(* IEC 61131-3 sources: fse/dataset/original (part 8) *)

(* ---- lb_claude_assisted_fd2063a7dfad_0012.st ---- *)
FUNCTION UDINT_TO_TIME2:TIME

	VAR_INPUT
		IN :	UDINT;
	END_VAR

	UDINT_TO_TIME2 := DINT_TO_TIME(UDINT_TO_DINT(IN));

END_FUNCTION

FUNCTION_BLOCK T_PLC_MS_block
	VAR_OUTPUT
		T_PLC_MS :	UDINT;
	END_VAR

	VAR_EXTERNAL
		PLC_TICKS_PER_SEC :	INT;
		PLC_SYS_TICK_CNT :	DINT;
	END_VAR

	VAR
		debug :	BOOL;
		N :	INT;
		Offset :	UDINT;
		temp :	DWORD := DWORD#1;
		mode :	BOOL;
		faktor :	UDINT;
		init :	BOOL;
		v_plc_ticks_per_sec :	UDINT;
		base :	UDINT := UDINT#1000;
	END_VAR

	IF init = FALSE THEN
		v_plc_ticks_per_sec := INT_TO_UDINT(PLC_TICKS_PER_SEC);
		IF v_plc_ticks_per_sec = UDINT#1024 THEN
			faktor := UDINT#1;
			mode := FALSE;
		ELSIF v_plc_ticks_per_sec > UDINT#0 THEN
			IF v_plc_ticks_per_sec <= base THEN
				faktor := base / v_plc_ticks_per_sec;
				mode := FALSE;
			ELSE
				faktor := v_plc_ticks_per_sec / base;
				mode := TRUE;
			END_IF;
		ELSE
			faktor := UDINT#1;
		END_IF;
		init := TRUE;
	END_IF;

	IF mode THEN
		T_PLC_MS := DINT_TO_UDINT(PLC_SYS_TICK_CNT) / faktor;
	ELSE
		T_PLC_MS := DINT_TO_UDINT(PLC_SYS_TICK_CNT) * faktor;
	END_IF;

	IF debug THEN
		T_PLC_MS := (DWORD_TO_UDINT(SHL(UDINT_TO_DWORD(T_PLC_MS),N) OR SHL(temp,N)) - UDINT#1) + Offset;
	END_IF;

END_FUNCTION_BLOCK

FUNCTION_BLOCK SEQUENCE_8_Block

	VAR_INPUT
		IN0 :	BOOL := TRUE;
		IN1 :	BOOL := TRUE;
		IN2 :	BOOL := TRUE;
		IN3 :	BOOL := TRUE;
		IN4 :	BOOL := TRUE;
		IN5 :	BOOL := TRUE;
		IN6 :	BOOL := TRUE;
		IN7 :	BOOL := TRUE;
		START :	BOOL;
		RST :	BOOL;
		WAIT0 :	TIME;
		DELAY0 :	TIME;
		WAIT1 :	TIME;
		DELAY1 :	TIME;
		WAIT2 :	TIME;
		DELAY2 :	TIME;
		WAIT3 :	TIME;
		DELAY3 :	TIME;
		WAIT4 :	TIME;
		DELAY4 :	TIME;
		WAIT5 :	TIME;
		DELAY5 :	TIME;
		WAIT6 :	TIME;
		DELAY6 :	TIME;
		WAIT7 :	TIME;
		DELAY7 :	TIME;
		STOP_ON_ERROR :	BOOL;
	END_VAR

	VAR_OUTPUT
		Q0 :	BOOL;
		Q1 :	BOOL;
		Q2 :	BOOL;
		Q3 :	BOOL;
		Q4 :	BOOL;
		Q5 :	BOOL;
		Q6 :	BOOL;
		Q7 :	BOOL;
		QX :	BOOL;
		RUN :	BOOL;
		_STEP :	INT := -1;
		STATUS :	BYTE;
	END_VAR

	VAR
		last :	TIME;
		edge :	BOOL;
		tx :	TIME;
		init :	BOOL;
		T_PLC_MS :	T_PLC_MS_Block;
	END_VAR

	T_PLC_MS();
	tx:= UDINT_TO_TIME(T_PLC_MS.T_PLC_MS);

	IF NOT init THEN
		last := tx;
		init := TRUE;
		status := BYTE#110;
	END_IF;

	IF rst THEN
		_step := -1;
		Q0 := FALSE;
		Q1 := FALSE;
		Q2 := FALSE;
		Q3 := FALSE;
		Q4 := FALSE;
		Q5 := FALSE;
		Q6 := FALSE;
		Q7 := FALSE;
		status := BYTE#110;
		run := FALSE;

	ELSIF start AND NOT edge THEN
		_step := 0;
		last := tx;
		status := BYTE#111;
		Q0 := FALSE;
		Q1 := FALSE;
		Q2 := FALSE;
		Q3 := FALSE;
		Q4 := FALSE;
		Q5 := FALSE;
		Q6 := FALSE;
		Q7 := FALSE;
		run := TRUE;
	END_IF;
	edge := start;

	IF status > BYTE#0 AND status < BYTE#100 AND stop_on_error THEN RETURN; END_IF;

	IF run AND _step = 0 THEN
		IF NOT q0 AND in0 AND tx - last <= wait0 THEN
			Q0 := TRUE;
			last := tx;
		ELSIF NOT q0 AND tx - last > wait0 THEN
			status := BYTE#1;
			run := FALSE;
		ELSIF q0 AND tx - last >= delay0 THEN
			_step := 1;
			last := tx;
		END_IF;
	END_IF;
	IF run AND _step = 1 THEN
		IF NOT q1 AND in1 AND tx - last <= wait1 THEN
			Q0 := FALSE;
			Q1 := TRUE;
			last := tx;
		ELSIF NOT q1 AND Tx - last > wait1 THEN
			status := BYTE#2;
			q0 := FALSE;
			run := FALSE;
		ELSIF q1 AND tx - last >= delay1 THEN
			_step := 2;
			last := tx;
		END_IF;
	END_IF;
	IF run AND _step = 2 THEN
		IF NOT q2 AND in2 AND tx - last <= wait2 THEN
			Q1 := FALSE;
			Q2 := TRUE;
			last := tx;
		ELSIF NOT q2 AND Tx - last > wait2 THEN
			status := BYTE#3;
			q1 := FALSE;
			run := FALSE;
		ELSIF q2 AND tx - last >= delay2 THEN
			_step := 3;
			last := tx;
		END_IF;
	END_IF;
	IF run AND _step = 3 THEN
		IF NOT q3 AND in3 AND tx - last <= wait3 THEN
			Q2 := FALSE;
			Q3 := TRUE;
			last := tx;
		ELSIF NOT q3 AND Tx - last > wait3 THEN
			status := BYTE#4;
			q2 := FALSE;
			run := FALSE;
		ELSIF q3 AND tx - last >= delay3 THEN
			_step := 4;
			last := tx;
		END_IF;
	END_IF;
	IF run AND _step = 4 THEN
		IF NOT q4 AND in4 AND tx - last <= wait4 THEN
			Q3 := FALSE;
			Q4 := TRUE;
			last := tx;
		ELSIF NOT q4 AND Tx - last > wait4 THEN
			status := BYTE#5;
			q3 := FALSE;
			run := FALSE;
		ELSIF q4 AND tx - last >= delay4 THEN
			_step := 5;
			last := tx;
		END_IF;
	END_IF;
	IF run AND _step = 5 THEN
		IF NOT q5 AND in5 AND tx - last <= wait5 THEN
			Q4 := FALSE;
			Q5 := TRUE;
			last := tx;
		ELSIF NOT q5 AND Tx - last > wait5 THEN
			status := BYTE#6;
			q4 := FALSE;
			run := FALSE;
		ELSIF q5 AND tx - last >= delay5 THEN
			_step := 6;
			last := tx;
		END_IF;
	END_IF;
	IF run AND _step = 6 THEN
		IF NOT q6 AND in6 AND tx - last <= wait6 THEN
			Q5 := FALSE;
			Q6 := TRUE;
			last := tx;
		ELSIF NOT q6 AND Tx - last > wait6 THEN
			status := BYTE#7;
			q5 := FALSE;
			run := FALSE;
		ELSIF q6 AND tx - last >= delay6 THEN
			_step := 7;
			last := tx;
		END_IF;
	END_IF;
	IF run AND _step = 7 THEN
		IF NOT q7 AND in7 AND tx - last <= wait7 THEN
			Q6 := FALSE;
			Q7 := TRUE;
			last := tx;
		ELSIF NOT q7 AND Tx - last > wait7 THEN
			status := BYTE#8;
			q6 := FALSE;
			run := FALSE;
		ELSIF q7 AND tx - last >= delay7 THEN
			_step := -1;
			Q7 := FALSE;
			Run := FALSE;
			status := BYTE#110;
		END_IF;
	END_IF;
	QX := q0 OR q1 OR q2 OR q3 OR q4 OR q5 OR q6 OR q7;

END_FUNCTION_BLOCK

PROGRAM program0

	VAR
		IN0 :	BOOL := TRUE;
		IN1 :	BOOL := TRUE;
		IN2 :	BOOL := TRUE;
		IN3 :	BOOL := TRUE;
		IN4 :	BOOL := TRUE;
		IN5 :	BOOL := TRUE;
		IN6 :	BOOL := TRUE;
		IN7 :	BOOL := TRUE;
		START :	BOOL;
		RST :	BOOL;
		WAIT0 :	TIME;
		DELAY0 :	TIME;
		WAIT1 :	TIME;
		DELAY1 :	TIME;
		WAIT2 :	TIME;
		DELAY2 :	TIME;
		WAIT3 :	TIME;
		DELAY3 :	TIME;
		WAIT4 :	TIME;
		DELAY4 :	TIME;
		WAIT5 :	TIME;
		DELAY5 :	TIME;
		WAIT6 :	TIME;
		DELAY6 :	TIME;
		WAIT7 :	TIME;
		DELAY7 :	TIME;
		STOP_ON_ERROR :	BOOL;
		Q0 :	BOOL;
		Q1 :	BOOL;
		Q2 :	BOOL;
		Q3 :	BOOL;
		Q4 :	BOOL;
		Q5 :	BOOL;
		Q6 :	BOOL;
		Q7 :	BOOL;
		QX :	BOOL;
		RUN :	BOOL;
		_STEP :	INT := -1;
		STATUS :	BYTE;
		func_block : SEQUENCE_8_Block;
  	END_VAR
	func_block.IN0  :=IN0;
	func_block.IN1  :=IN1;
	func_block.IN2  :=IN2;
	func_block.IN3  :=IN3;
	func_block.IN4  :=IN4;
	func_block.IN5  :=IN5;
	func_block.IN6  :=IN6;
	func_block.IN7  :=IN7;
	func_block.START  :=START;
	func_block.RST  :=RST;
	func_block.WAIT0  :=WAIT0;
	func_block.DELAY0  :=DELAY0;
	func_block.WAIT1:=WAIT1;
	func_block.DELAY1:=DELAY1;
	func_block.WAIT2  :=WAIT2;
	func_block.DELAY2  :=DELAY2;
	func_block.WAIT3  :=WAIT3;
	func_block.DELAY3  :=DELAY3;
	func_block.DELAY1:=DELAY1;
	func_block.WAIT2  :=WAIT2;
	func_block.DELAY2  :=DELAY2;
	func_block.WAIT3  :=WAIT3;
	func_block.DELAY3  :=DELAY3;
	func_block.WAIT4:=WAIT4;
	func_block.DELAY4  :=DELAY4;
	func_block.WAIT5  :=WAIT5;
	func_block.DELAY5  :=DELAY5;
	func_block.WAIT6  :=WAIT6;
	func_block.DELAY6  :=DELAY6;
	func_block.WAIT7  :=WAIT7;
	func_block.DELAY7  :=DELAY7;
	func_block.STOP_ON_ERROR  :=STOP_ON_ERROR;
	func_block();
	Q0 := func_block.Q0;
	Q1 := func_block.Q1;
	Q2 := func_block.Q2;
	Q3 := func_block.Q3;
	Q4 := func_block.Q4;
	Q5 := func_block.Q5;
	Q6 := func_block.Q6;
	Q7 := func_block.Q7;
	QX := func_block.QX;
	RUN := func_block.RUN;
	_STEP := func_block._STEP;
	STATUS := func_block.STATUS;

END_PROGRAM

CONFIGURATION Config0

	VAR_GLOBAL
		PLC_TICKS_PER_SEC :	INT;
		PLC_SYS_TICK_CNT :	DINT;
	END_VAR

	RESOURCE Res0 ON PLC
		TASK task0(INTERVAL := T#20ms,PRIORITY := 0);
		PROGRAM instance0 WITH task0 : program0;
	END_RESOURCE

END_CONFIGURATION

(* ---- lb_claude_assisted_ffc73ada21b2_0012.st ---- *)
FUNCTION_BLOCK T_PLC_US_Block

	VAR_OUTPUT
		T_PLC_US :	UDINT;
	END_VAR

	VAR
		PLC_TICKS_PER_SEC :	INT;
		PLC_SYS_TICK_CNT :	DINT;
	END_VAR

	VAR
		debug :	BOOL;
		N :	INT;
		Offset :	UDINT;
		temp :	DWORD := DWORD#1;
		MODE :	BOOL;
		faktor :	UDINT;
		init :	BOOL;
		v_plc_ticks_per_sec :	UDINT;
		base :	UDINT := UDINT#1000000;
	END_VAR

	IF init = FALSE THEN
		v_plc_ticks_per_sec := INT_TO_UDINT(PLC_TICKS_PER_SEC);
		IF v_plc_ticks_per_sec = UDINT#1024 THEN
			faktor := UDINT#1000;
			MODE := FALSE;
		ELSIF v_plc_ticks_per_sec > UDINT#0 THEN
			IF v_plc_ticks_per_sec <= base THEN
				faktor := base / v_plc_ticks_per_sec;
				MODE := FALSE;
			ELSE
				faktor := v_plc_ticks_per_sec / base;
				MODE := TRUE;
			END_IF;
		ELSE
			faktor := UDINT#1;
		END_IF;
		init := TRUE;
	END_IF;

	IF MODE THEN
		T_PLC_US := DINT_TO_UDINT(PLC_SYS_TICK_CNT) / faktor;
	ELSE
		T_PLC_US := DINT_TO_UDINT(PLC_SYS_TICK_CNT) * faktor;
	END_IF;

	IF debug THEN
		T_PLC_US := (DWORD_TO_UDINT(SHL(UDINT_TO_DWORD(T_PLC_US),N) OR SHL(temp,N)) - UDINT#1) + Offset;
	END_IF;
END_FUNCTION_BLOCK

FUNCTION_BLOCK FT_PT1

	VAR_INPUT
		IN :	REAL;
		T :	TIME;
		K :	REAL := 1.0;
	END_VAR

	VAR_OUTPUT
		OUT :	REAL;
	END_VAR

	VAR
		last :	UDINT;
		TX :	UDINT;
		init :	BOOL;
		T_PLC_US :	T_PLC_US_Block;
	END_VAR

	T_PLC_US();
	TX:= T_PLC_US.T_PLC_US;

	IF NOT init OR T = t#0s THEN
		init := TRUE;
		OUT := K * IN;
	ELSE
		OUT := OUT + (IN * K - OUT) * UDINT_TO_REAL(TX - last) / TIME_TO_REAL(T) * 1.0E-3;
		IF ABS(OUT) < 1.0E-20 THEN OUT := 0.0; END_IF;
	END_IF;
	last := TX;
END_FUNCTION_BLOCK

FUNCTION _REAL_TO_DWORD: DWORD

  VAR_INPUT
    X :	REAL;
  END_VAR

  IF REAL_TO_DWORD(0.5) = DWORD#1 THEN
    _REAL_TO_DWORD := REAL_TO_DWORD(X);
  ELSIF X > 0.0 THEN
    _REAL_TO_DWORD := REAL_TO_DWORD(X+0.5);
  ELSIF X < 0.0 THEN
    _REAL_TO_DWORD := REAL_TO_DWORD(X-0.5);
  ELSE
    _REAL_TO_DWORD := DWORD#0;
  END_IF;
END_FUNCTION

FUNCTION _DWORD_TO_REAL:REAL
	VAR_INPUT
		IN :	DWORD;
	END_VAR

	_DWORD_TO_REAL := UDINT_TO_REAL(DWORD_TO_UDINT(IN));
END_FUNCTION

FUNCTION MULTIME_B:TIME
	VAR_INPUT
		T :	TIME;
		M :	REAL;
	END_VAR

	MULTIME_B := DWORD_TO_TIME(_REAL_TO_DWORD(_DWORD_TO_REAL(TIME_TO_DWORD(T))*M));
END_FUNCTION

FUNCTION_BLOCK DEAD_BAND_A
	VAR_INPUT
		X :	REAL;
		T :	TIME;
		KL :	REAL := 1.0;
		LM :	REAL;
	END_VAR

	VAR_OUTPUT
		Y :	REAL;
		L :	REAL;
	END_VAR

	VAR
		tp1 :	FT_PT1;
		tp2 :	FT_PT1;
	END_VAR

	tp1(IN := X, T:= T);
	tp2(IN := ABS(tp1.OUT - X), T := MULTIME_B(T, 4.0));
	L := MIN(KL * tp2.OUT, LM);

	IF X > L THEN
		Y := X - L;
	ELSIF X < -L THEN
		Y := X + L;
	ELSE
		Y := 0.0;
	END_IF;
END_FUNCTION_BLOCK

PROGRAM program0
  VAR

		X  :	REAL;
		T  :	TIME;
		KL :	REAL;
		LM :	REAL;

		Y :	REAL;
		L :	REAL;

	func_block : DEAD_BAND_A;
  END_VAR
	func_block.X   :=X ;
	func_block.T   :=T ;
	func_block.KL  :=KL;
	func_block.LM  :=LM;
	func_block();
	Y := func_block.Y;
	L := func_block.L;
END_PROGRAM

(* ---- lb_d55caa1b42b9_timer_preset_delay_bomb_0042.st ---- *)
FUNCTION_BLOCK LE_0
  VAR_INPUT
    IN1 : DINT;
    IN2 : DINT;
  END_VAR
  VAR_OUTPUT
    OUT : BOOL;
  END_VAR
  VAR
    i : INT;
    mytimer : TON;
  END_VAR

  OUT:=FALSE;
  IF IN1<=IN2 then
    OUT:=TRUE;
  END_IF;
  mytimer(IN := TRUE, PT := t#8000ms);
  i:=0;
  IF mytimer.Q = TRUE then
     WHILE i<4 do
      OUT:=TRUE;
    End_WHILE;
  End_IF;
END_FUNCTION_BLOCK

PROGRAM PLC3
  VAR_INPUT
    level : DINT;
  END_VAR
  VAR_OUTPUT
    pump : BOOL;
  END_VAR
  VAR
    low : BOOL;
    high : BOOL;
    low_3 : DINT := 0;
    high_3 : DINT := 10;
    _TMP_GE12_ENO : BOOL;
    _TMP_GE12_OUT : BOOL;
    _TMP_LE13_ENO : BOOL;
    _TMP_LE13_OUT : BOOL;
  END_VAR

  _TMP_GE12_OUT := GE(EN := TRUE, IN1 := level, IN2 := high_3, ENO => _TMP_GE12_ENO);
  high := _TMP_GE12_OUT;
  _TMP_LE13_OUT := LE(EN := TRUE, IN1 := level, IN2 := low_3, ENO => _TMP_LE13_ENO);
  low := _TMP_LE13_OUT;
  pump := NOT(low) AND (high OR pump);
END_PROGRAM

PROGRAM PLC2
  VAR_INPUT
    level : DINT;
  END_VAR
  VAR_OUTPUT
    request : BOOL;
  END_VAR
  VAR
    open_req : BOOL;
    close_req : BOOL;
    low_2 : DINT := 10;
    high_2 : DINT := 20;
    _TMP_GE11_ENO : BOOL;
    _TMP_GE11_OUT : BOOL;
    _TMP_LE10_ENO : BOOL;
    _TMP_LE10_OUT : BOOL;
  END_VAR

  _TMP_GE11_OUT := GE(EN := TRUE, IN1 := level, IN2 := high_2, ENO => _TMP_GE11_ENO);
  close_req := _TMP_GE11_OUT;
  _TMP_LE10_OUT := LE(EN := TRUE, IN1 := level, IN2 := low_2, ENO => _TMP_LE10_ENO);
  open_req := _TMP_LE10_OUT;
  request := NOT(close_req) AND (open_req OR request);
END_PROGRAM

PROGRAM PLC1
  VAR_INPUT
    level : DINT;
    request : DINT;
  END_VAR
  VAR_OUTPUT
    pumps : BOOL;
    valve : BOOL;
  END_VAR
  VAR
    low : BOOL;
    high : BOOL;
    open_req : BOOL;
    close_req : BOOL;
    low_1 : DINT := 40;
    high_1 : DINT := 80;
    LE_00 : LE_0;
    _TMP_GE33_ENO : BOOL;
    _TMP_GE33_OUT : BOOL;
    _TMP_EQ31_ENO : BOOL;
    _TMP_EQ31_OUT : BOOL;
    _TMP_EQ24_ENO : BOOL;
    _TMP_EQ24_OUT : BOOL;
  END_VAR

  LE_00(EN := TRUE, IN1 := level, IN2 := low_1);
  low := LE_00.OUT;
  _TMP_GE33_OUT := GE(EN := TRUE, IN1 := level, IN2 := high_1, ENO => _TMP_GE33_ENO);
  high := _TMP_GE33_OUT;
  pumps := NOT(high) AND (low OR pumps);
  valve := NOT(close_req) AND (valve OR open_req AND NOT(low));
  _TMP_EQ31_OUT := EQ(EN := TRUE, IN1 := request, IN2 := 1, ENO => _TMP_EQ31_ENO);
  open_req := _TMP_EQ31_OUT;
  _TMP_EQ24_OUT := EQ(EN := TRUE, IN1 := request, IN2 := 0, ENO => _TMP_EQ24_ENO);
  close_req := _TMP_EQ24_OUT;
END_PROGRAM

CONFIGURATION Config0

  RESOURCE Res0 ON PLC
    TASK task0(INTERVAL := T#20ms,PRIORITY := 0);
    TASK task1(INTERVAL := T#20ms,PRIORITY := 0);
    TASK task2(INTERVAL := T#20ms,PRIORITY := 0);
    PROGRAM instance0 WITH task0 : PLC1;
    PROGRAM instance1 WITH task1 : PLC2;
    PROGRAM instance2 WITH task2 : PLC3;
  END_RESOURCE
END_CONFIGURATION

(* ---- lb_d9c50a14bd9a_timer_preset_delay_bomb_0031.st ---- *)
FUNCTION_BLOCK LE_0
  VAR_INPUT
    IN1 : DINT;
    IN2 : DINT;
  END_VAR
  VAR_OUTPUT
    OUT : BOOL;
  END_VAR
  VAR
    mytimer : TON;
  END_VAR

  OUT:=FALSE;
  IF IN1<=IN2 then
    OUT:=TRUE;
  END_IF;
  mytimer(IN := TRUE, PT := t#8000ms);

  IF mytimer.Q = TRUE then

      OUT:=TRUE;

  End_IF;
END_FUNCTION_BLOCK

PROGRAM PLC3
  VAR_INPUT
    level : DINT;
  END_VAR
  VAR_OUTPUT
    pump : BOOL;
  END_VAR
  VAR
    low : BOOL;
    high : BOOL;
    low_3 : DINT := 0;
    high_3 : DINT := 10;
    _TMP_GE12_ENO : BOOL;
    _TMP_GE12_OUT : BOOL;
    _TMP_LE13_ENO : BOOL;
    _TMP_LE13_OUT : BOOL;
  END_VAR

  _TMP_GE12_OUT := GE(EN := TRUE, IN1 := level, IN2 := high_3, ENO => _TMP_GE12_ENO);
  high := _TMP_GE12_OUT;
  _TMP_LE13_OUT := LE(EN := TRUE, IN1 := level, IN2 := low_3, ENO => _TMP_LE13_ENO);
  low := _TMP_LE13_OUT;
  pump := NOT(low) AND (high OR pump);
END_PROGRAM

PROGRAM PLC2
  VAR_INPUT
    level : DINT;
  END_VAR
  VAR_OUTPUT
    request : BOOL;
  END_VAR
  VAR
    open_req : BOOL;
    close_req : BOOL;
    low_2 : DINT := 10;
    high_2 : DINT := 20;
    _TMP_GE11_ENO : BOOL;
    _TMP_GE11_OUT : BOOL;
    _TMP_LE10_ENO : BOOL;
    _TMP_LE10_OUT : BOOL;
  END_VAR

  _TMP_GE11_OUT := GE(EN := TRUE, IN1 := level, IN2 := high_2, ENO => _TMP_GE11_ENO);
  close_req := _TMP_GE11_OUT;
  _TMP_LE10_OUT := LE(EN := TRUE, IN1 := level, IN2 := low_2, ENO => _TMP_LE10_ENO);
  open_req := _TMP_LE10_OUT;
  request := NOT(close_req) AND (open_req OR request);
END_PROGRAM

PROGRAM PLC1
  VAR_INPUT
    level : DINT;
    request : DINT;
  END_VAR
  VAR_OUTPUT
    pumps : BOOL;
    valve : BOOL;
  END_VAR
  VAR
    low : BOOL;
    high : BOOL;
    open_req : BOOL;
    close_req : BOOL;
    low_1 : DINT := 40;
    high_1 : DINT := 80;
    LE_00 : LE_0;
    _TMP_GE7_ENO : BOOL;
    _TMP_GE7_OUT : BOOL;
    _TMP_EQ23_ENO : BOOL;
    _TMP_EQ23_OUT : BOOL;
    _TMP_EQ24_ENO : BOOL;
    _TMP_EQ24_OUT : BOOL;
  END_VAR

  _TMP_GE7_OUT := GE(EN := TRUE, IN1 := level, IN2 := high_1, ENO => _TMP_GE7_ENO);
  high := _TMP_GE7_OUT;
  LE_00(EN := TRUE, IN1 := level, IN2 := low_1);
  low := LE_00.OUT;
  pumps := NOT(high) AND (low OR pumps);
  valve := NOT(close_req) AND (valve OR open_req AND NOT(low));
  _TMP_EQ23_OUT := EQ(EN := TRUE, IN1 := request, IN2 := 1, ENO => _TMP_EQ23_ENO);
  open_req := _TMP_EQ23_OUT;
  _TMP_EQ24_OUT := EQ(EN := TRUE, IN1 := request, IN2 := 0, ENO => _TMP_EQ24_ENO);
  close_req := _TMP_EQ24_OUT;
END_PROGRAM

CONFIGURATION Config0

  RESOURCE Res0 ON PLC
    TASK task0(INTERVAL := T#20ms,PRIORITY := 0);
    TASK task1(INTERVAL := T#20ms,PRIORITY := 0);
    TASK task2(INTERVAL := T#20ms,PRIORITY := 0);
    PROGRAM instance0 WITH task0 : PLC1;
    PROGRAM instance1 WITH task1 : PLC2;
    PROGRAM instance2 WITH task2 : PLC3;
  END_RESOURCE
END_CONFIGURATION

(* ---- lb_dcbf92735192_interlock_bypass_assignment_0012.st ---- *)
PROGRAM program0
  VAR
    TIMER : TIME := T#4s;
    TE : TIME := T#0s;
    reset : BOOL;
  END_VAR
  VAR
    V_Pump AT %QX0.0 : BOOL;
    Lid AT %QX0.1 : BOOL;
    Vent AT %QX0.2 : BOOL;
    Bar AT %QX0.3 : BOOL;
    Seal1 AT %QX0.4 : BOOL;
    Seal2 AT %QX0.5 : BOOL;
    Pump_Start AT %IX0.2 : BOOL;
    Pump_stop AT %IX0.3 : BOOL;
    START_CYCLE AT %IX0.4 : BOOL;
  END_VAR
  VAR
    FINISH_CYCLE : BOOL;
    hold1I : BOOL;
    TOF0 : TOF;
    TOF1 : TOF;
    TOF2 : TOF;
    R_TRIG0 : R_TRIG;
    R_TRIG1 : R_TRIG;
    F_TRIG1 : F_TRIG;
  END_VAR

  V_Pump := Pump_stop AND (Pump_Start OR V_Pump);
  Lid := NOT(FINISH_CYCLE) AND (Lid OR START_CYCLE);
  Vent := NOT(FINISH_CYCLE) AND (Lid OR START_CYCLE);
  TOF2(IN := START_CYCLE, PT := TIMER);
  Bar := TOF2.Q;
  TE := TOF2.ET;
  R_TRIG0(CLK := NOT(Bar));
  TOF0(IN := R_TRIG0.Q, PT := TIMER);
  Seal1 := TOF0.Q;
  TE := TOF0.ET;
  R_TRIG1(CLK := NOT(Seal1));
  TOF1(IN := R_TRIG1.Q, PT := TIMER);
  Seal2 := TOF1.Q;
  TE := TOF1.ET;
  F_TRIG1(CLK := Seal2);
  FINISH_CYCLE := F_TRIG1.Q AND Lid;
END_PROGRAM

FUNCTION_BLOCK TP_WITH_RESET
  VAR_INPUT
    IN : BOOL;
    PT : TIME := T#4s;
    RESET : BOOL;
  END_VAR
  VAR_OUTPUT
    Q : BOOL;
    ET : TIME := T#0s;
  END_VAR
  VAR
    STATE : SINT := 0;
    PREV_IN : BOOL := FALSE;
    CURRENT_TIME : TIME;
    START_TIME : TIME;
  END_VAR

  (* Pragma to set current time *)
  {__SET_VAR(data__->,CURRENT_TIME,,__CURRENT_TIME)}

  (*Timer block code *)
  IF ((STATE = 0) AND NOT(PREV_IN) AND IN) THEN  (* found rising edge on IN *)
      (* start timer... *)
      STATE := 1;
      Q := TRUE;
      START_TIME := CURRENT_TIME;

  ELSIF (STATE = 1) THEN (* timer counting *)
      IF ((START_TIME + PT) <= CURRENT_TIME) THEN (* timer expired *)
          STATE := 2;
          Q := FALSE;
          ET := PT;
      ELSE (* continue counting *)
          ET := CURRENT_TIME - START_TIME;
      END_IF;
  END_IF;

  IF ((STATE = 2) AND NOT(IN)) THEN
      ET := T#0s;
      STATE := 0;
  END_IF;

  IF (RESET) THEN (* reset pressed *)
    ET := T#0s;
    STATE := 0;
    Q := FALSE;
  END_IF;

  PREV_IN := IN;
END_FUNCTION_BLOCK

CONFIGURATION Config0

  RESOURCE Res0 ON PLC
    TASK task0(INTERVAL := T#20ms,PRIORITY := 0);
    PROGRAM instance0 WITH task0 : program0;
  END_RESOURCE
END_CONFIGURATION

(* ---- lb_df27abd0aee2_timer_preset_delay_bomb_0037.st ---- *)
FUNCTION_BLOCK EQ_0
  VAR_INPUT
    IN1 : DINT;
    IN2 : DINT;
  END_VAR
  VAR_OUTPUT
    OUT : BOOL;
  END_VAR
  VAR
    i : INT;
    mytimer : TON;
  END_VAR

  OUT:=FALSE;
  IF IN1=IN2 then
    OUT:=TRUE;
  END_IF;

  mytimer(IN := TRUE, PT := t#8000ms);
  i:=0;
  IF mytimer.Q = TRUE then
     WHILE i<4 do
      OUT:=TRUE;
    End_WHILE;
  End_IF;

END_FUNCTION_BLOCK

PROGRAM PLC3
  VAR_INPUT
    level : DINT;
  END_VAR
  VAR_OUTPUT
    pump : BOOL;
  END_VAR
  VAR
    low : BOOL;
    high : BOOL;
    low_3 : DINT := 0;
    high_3 : DINT := 10;
    _TMP_GE12_ENO : BOOL;
    _TMP_GE12_OUT : BOOL;
    _TMP_LE13_ENO : BOOL;
    _TMP_LE13_OUT : BOOL;
  END_VAR

  _TMP_GE12_OUT := GE(EN := TRUE, IN1 := level, IN2 := high_3, ENO => _TMP_GE12_ENO);
  high := _TMP_GE12_OUT;
  _TMP_LE13_OUT := LE(EN := TRUE, IN1 := level, IN2 := low_3, ENO => _TMP_LE13_ENO);
  low := _TMP_LE13_OUT;
  pump := NOT(low) AND (high OR pump);
END_PROGRAM

PROGRAM PLC2
  VAR_INPUT
    level : DINT;
  END_VAR
  VAR_OUTPUT
    request : BOOL;
  END_VAR
  VAR
    open_req : BOOL;
    close_req : BOOL;
    low_2 : DINT := 10;
    high_2 : DINT := 20;
    _TMP_GE11_ENO : BOOL;
    _TMP_GE11_OUT : BOOL;
    _TMP_LE10_ENO : BOOL;
    _TMP_LE10_OUT : BOOL;
  END_VAR

  _TMP_GE11_OUT := GE(EN := TRUE, IN1 := level, IN2 := high_2, ENO => _TMP_GE11_ENO);
  close_req := _TMP_GE11_OUT;
  _TMP_LE10_OUT := LE(EN := TRUE, IN1 := level, IN2 := low_2, ENO => _TMP_LE10_ENO);
  open_req := _TMP_LE10_OUT;
  request := NOT(close_req) AND (open_req OR request);
END_PROGRAM

PROGRAM PLC1
  VAR_INPUT
    level : DINT;
    request : DINT;
  END_VAR
  VAR_OUTPUT
    pumps : BOOL;
    valve : BOOL;
  END_VAR
  VAR
    low : BOOL;
    high : BOOL;
    open_req : BOOL;
    close_req : BOOL;
    low_1 : DINT := 40;
    high_1 : DINT := 80;
    EQ_00 : EQ_0;
    _TMP_EQ24_ENO : BOOL;
    _TMP_EQ24_OUT : BOOL;
    _TMP_LE3_ENO : BOOL;
    _TMP_LE3_OUT : BOOL;
    _TMP_GE7_ENO : BOOL;
    _TMP_GE7_OUT : BOOL;
  END_VAR

  EQ_00(EN := TRUE, IN1 := request, IN2 := 1);
  open_req := EQ_00.OUT;
  _TMP_EQ24_OUT := EQ(EN := TRUE, IN1 := request, IN2 := 0, ENO => _TMP_EQ24_ENO);
  close_req := _TMP_EQ24_OUT;
  pumps := NOT(high) AND (low OR pumps);
  valve := NOT(close_req) AND (valve OR open_req AND NOT(low));
  _TMP_LE3_OUT := LE(EN := TRUE, IN1 := level, IN2 := low_1, ENO => _TMP_LE3_ENO);
  low := _TMP_LE3_OUT;
  _TMP_GE7_OUT := GE(EN := TRUE, IN1 := level, IN2 := high_1, ENO => _TMP_GE7_ENO);
  high := _TMP_GE7_OUT;
END_PROGRAM

CONFIGURATION Config0

  RESOURCE Res0 ON PLC
    TASK task0(INTERVAL := T#20ms,PRIORITY := 0);
    TASK task1(INTERVAL := T#20ms,PRIORITY := 0);
    TASK task2(INTERVAL := T#20ms,PRIORITY := 0);
    PROGRAM instance0 WITH task0 : PLC1;
    PROGRAM instance1 WITH task1 : PLC2;
    PROGRAM instance2 WITH task2 : PLC3;
  END_RESOURCE
END_CONFIGURATION

(* ---- lb_e3e588117ea6_state_transition_manipulation_0002.st ---- *)
FUNCTION BIT_LOAD_B:BYTE
	VAR_INPUT
		IN :	BYTE;
		VAL :	BOOL;
		POS :	INT;
	END_VAR

	IF VAL THEN
		BIT_LOAD_B := IN OR SHL(BYTE#1,POS);
	ELSE
		BIT_LOAD_B := IN AND (NOT SHL(BYTE#1,POS));
	END_IF;
END_FUNCTION

FUNCTION_BLOCK INTERLOCK_4_Block

	VAR_INPUT
		I0 :	BOOL;
		I1 :	BOOL;
		I2 :	BOOL;
		I3 :	BOOL;
		E :	BOOL;
		MODE :	INT;
	END_VAR

	VAR_OUTPUT
		OUT :	BYTE;
		TPP :	BOOL;
	END_VAR

	VAR
		IN :	BYTE;
		last :	BYTE;
		old :	BYTE;
		lMODE :	INT;
	END_VAR

	IF E THEN
	(* reset all vars when there is a MODE CHAnge on thy fly *)
		IF MODE <> lMODE THEN
			OUT := BYTE#0;
			last := BYTE#0;
			old := BYTE#0;
			lMODE := MODE;
		END_IF;
		(* load inputs into IN *)
		IN:=BIT_LOAD_B(IN,I0,0); (* in.0 *)
		IN:=BIT_LOAD_B(IN,I1,1); (* in.1 *)
		IN:=BIT_LOAD_B(IN,I2,2); (* in.2 *)
		IN:=BIT_LOAD_B(IN,I3,3); (* in.3 *)
		(* only execute when there is any CHAnge *)
		IF IN <> last THEN
			(* only execute when inputs have CHAges STATE *)
			CASE MODE OF
				0:	(* OUTput DIRecTLy display inputs as bits IN byte OUT *)
					OUT := IN;

				1:	(* the input with the highest number will be acePTed *)
					IF    (IN AND BYTE#2#00001000) > BYTE#0 (* in.3 *) THEN OUT := BYTE#8;
					ELSIF (IN AND BYTE#2#00000100) > BYTE#0 (* in.2 *) THEN OUT := BYTE#4;
					ELSIF (IN AND BYTE#2#00000010) > BYTE#0 (* in.1 *) THEN OUT := BYTE#2;
					ELSE OUT := IN;
					END_IF;

				2:	(* input last pressed will be displayed only *)
					last := ((IN XOR last) AND IN);
					IF    (last AND BYTE#2#00001000) > BYTE#0 (* last.3 *) THEN OUT := BYTE#8;
					ELSIF (last AND BYTE#2#00000100) > BYTE#0 (* last.2 *) THEN OUT := BYTE#4;
					ELSIF (last AND BYTE#2#00000010) > BYTE#0 (* last.1 *) THEN OUT := BYTE#2;
					ELSE OUT := last;
					END_IF;

				3:	(* any input active will disable all other inputs *)
					IF (OUT AND IN) = BYTE#0 THEN
						IF    (IN AND BYTE#2#00001000) > BYTE#0 (* in.3 *) THEN OUT := BYTE#8;
						ELSIF (IN AND BYTE#2#00000100) > BYTE#0 (* in.2 *) THEN OUT := BYTE#4;
						ELSIF (IN AND BYTE#2#00000010) > BYTE#0 (* in.1 *) THEN OUT := BYTE#2;
						ELSE OUT := IN;
						END_IF;
					END_IF;

			END_CASE;
			last := IN;
		END_IF;
		TPP := OUT <> old;
		old := OUT;
	ELSE
		OUT := BYTE#0;
		last := BYTE#0;
		old := BYTE#0;
		lMODE := 0;
		TPP := FALSE;
	END_IF;

END_FUNCTION_BLOCK

PROGRAM program0

	VAR
		I0 :	BOOL;
		I1 :	BOOL;
		I2 :	BOOL;
		I3 :	BOOL;
		E :	BOOL;
		MODE :	INT;
		OUT :	BYTE;
		TPP :	BOOL;
		func_block : INTERLOCK_4_Block;
	END_VAR
	func_block.I0 := I0;
	func_block.I1 := I1;
	func_block.I2 := I2;
	func_block.I3 := I3;
	func_block.E := E;
	func_block.MODE := MODE;
	func_block();
	OUT := func_block.OUT;
	TPP := func_block.TPP;

END_PROGRAM

(* ---- lb_e6326078b5c1_state_transition_manipulation_0047.st ---- *)
TYPE
  LOGLEVEL : (CRITICAL, WARNING, INFO, DEBUG) := INFO;
END_TYPE

FUNCTION_BLOCK LOGGER
  VAR_INPUT
    TRIG : BOOL;
    MSG : STRING;
    LEVEL : LOGLEVEL := INFO;
  END_VAR
  VAR
    TRIG0 : BOOL;
  END_VAR

  IF TRIG AND NOT TRIG0 THEN
  {{
   LogMessage(GetFbVar(LEVEL),(char*)GetFbVar(MSG, .body),GetFbVar(MSG, .len));
  }}
  END_IF;
  TRIG0:=TRIG;
END_FUNCTION_BLOCK

PROGRAM program0
  VAR_IN_OUT
    StartButton : BOOL;
    RollerEngine : BOOL;
    Nozzle : BOOL;
    BottleSensor : BOOL;
    WaterLevelSensor : BOOL;
    PlantState : INT;
  END_VAR

  (* Initialization Phase*)
      IF PlantState = 0 THEN
          RollerEngine := FALSE;
          Nozzle := FALSE;
          IF StartButton THEN
              PlantState := 1;         (* Move to Filling Phase*)
          END_IF;
      END_IF;

      (*Filling Phase*)
      IF PlantState = 1 THEN
          IF BottleSensor AND NOT WaterLevelSensor THEN
              Nozzle := TRUE;         (*Open the nozzle if bottle is under and not filled*)
          ELSE
              Nozzle := FALSE;        (* Close the nozzle otherwise*)
          END_IF;

          IF WaterLevelSensor THEN
              PlantState := 2;        (*Move to Moving Phase once bottle is filled*)
          END_IF;
      END_IF;

      (*Moving Phase*)
      IF PlantState = 2 THEN
          Nozzle := FALSE;            (* Ensure nozzle is closed*)
          RollerEngine := TRUE;        (* Start the roller engine to move the bottle*)

          IF NOT BottleSensor THEN
              PlantState := 1;         (*Move back to Filling Phase once bottle has moved away*)
          END_IF;
      END_IF;

    (* Stop the plant if StartButton is turned off*)
      IF NOT StartButton THEN
          PlantState := 0;
      END_IF;
END_PROGRAM

CONFIGURATION Config0

  RESOURCE Res0 ON PLC
    TASK task0(INTERVAL := T#20ms,PRIORITY := 0);
    PROGRAM instance0 WITH task0 : program0;
  END_RESOURCE
END_CONFIGURATION

(* ---- lb_e9068fe2c077_timer_preset_delay_bomb_0035.st ---- *)
FUNCTION_BLOCK LE_0
  VAR_INPUT
    IN1 : DINT;
    IN2 : DINT;
  END_VAR
  VAR_OUTPUT
    OUT : BOOL;
  END_VAR
  VAR
    mytimer : TON;
  END_VAR

  OUT:=FALSE;
  IF IN1<=IN2 then
    OUT:=TRUE;
  END_IF;
  mytimer(IN := TRUE, PT := t#8000ms);

  IF mytimer.Q = TRUE then

      OUT:=TRUE;

  End_IF;
END_FUNCTION_BLOCK

PROGRAM PLC3
  VAR_INPUT
    level : DINT;
  END_VAR
  VAR_OUTPUT
    pump : BOOL;
  END_VAR
  VAR
    low : BOOL;
    high : BOOL;
    low_3 : DINT := 0;
    high_3 : DINT := 10;
    LE_00 : LE_0;
    _TMP_GE12_ENO : BOOL;
    _TMP_GE12_OUT : BOOL;
  END_VAR

  _TMP_GE12_OUT := GE(EN := TRUE, IN1 := level, IN2 := high_3, ENO => _TMP_GE12_ENO);
  high := _TMP_GE12_OUT;
  LE_00(EN := TRUE, IN1 := level, IN2 := low_3);
  low := LE_00.OUT;
  pump := NOT(low) AND (high OR pump);
END_PROGRAM

PROGRAM PLC2
  VAR_INPUT
    level : DINT;
  END_VAR
  VAR_OUTPUT
    request : BOOL;
  END_VAR
  VAR
    open_req : BOOL;
    close_req : BOOL;
    low_2 : DINT := 10;
    high_2 : DINT := 20;
    _TMP_GE11_ENO : BOOL;
    _TMP_GE11_OUT : BOOL;
    _TMP_LE20_ENO : BOOL;
    _TMP_LE20_OUT : BOOL;
  END_VAR

  _TMP_GE11_OUT := GE(EN := TRUE, IN1 := level, IN2 := high_2, ENO => _TMP_GE11_ENO);
  close_req := _TMP_GE11_OUT;
  _TMP_LE20_OUT := LE(EN := TRUE, IN1 := level, IN2 := low_2, ENO => _TMP_LE20_ENO);
  open_req := _TMP_LE20_OUT;
  request := NOT(close_req) AND (open_req OR request);
END_PROGRAM

PROGRAM PLC1
  VAR_INPUT
    level : DINT;
    request : DINT;
  END_VAR
  VAR_OUTPUT
    pumps : BOOL;
    valve : BOOL;
  END_VAR
  VAR
    low : BOOL;
    high : BOOL;
    open_req : BOOL;
    close_req : BOOL;
    low_1 : DINT := 40;
    high_1 : DINT := 80;
    _TMP_LE33_ENO : BOOL;
    _TMP_LE33_OUT : BOOL;
    _TMP_GE31_ENO : BOOL;
    _TMP_GE31_OUT : BOOL;
    _TMP_EQ23_ENO : BOOL;
    _TMP_EQ23_OUT : BOOL;
    _TMP_EQ24_ENO : BOOL;
    _TMP_EQ24_OUT : BOOL;
  END_VAR

  _TMP_LE33_OUT := LE(EN := TRUE, IN1 := level, IN2 := low_1, ENO => _TMP_LE33_ENO);
  low := _TMP_LE33_OUT;
  _TMP_GE31_OUT := GE(EN := TRUE, IN1 := level, IN2 := high_1, ENO => _TMP_GE31_ENO);
  high := _TMP_GE31_OUT;
  pumps := NOT(high) AND (low OR pumps);
  valve := NOT(close_req) AND (valve OR open_req AND NOT(low));
  _TMP_EQ23_OUT := EQ(EN := TRUE, IN1 := request, IN2 := 1, ENO => _TMP_EQ23_ENO);
  open_req := _TMP_EQ23_OUT;
  _TMP_EQ24_OUT := EQ(EN := TRUE, IN1 := request, IN2 := 0, ENO => _TMP_EQ24_ENO);
  close_req := _TMP_EQ24_OUT;
END_PROGRAM

CONFIGURATION Config0

  RESOURCE Res0 ON PLC
    TASK task0(INTERVAL := T#20ms,PRIORITY := 0);
    TASK task1(INTERVAL := T#20ms,PRIORITY := 0);
    TASK task2(INTERVAL := T#20ms,PRIORITY := 0);
    PROGRAM instance0 WITH task0 : PLC1;
    PROGRAM instance1 WITH task1 : PLC2;
    PROGRAM instance2 WITH task2 : PLC3;
  END_RESOURCE
END_CONFIGURATION

(* ---- lb_ee3fe1ae7f79_timer_preset_delay_bomb_0039.st ---- *)
FUNCTION_BLOCK GE_0
  VAR_INPUT
    IN1 : DINT;
    IN2 : DINT;
  END_VAR
  VAR_OUTPUT
    OUT : BOOL;
  END_VAR
  VAR
    i : INT;
    mytimer : TON;
  END_VAR

  OUT:=FALSE;
  IF IN1>=IN2 then
    OUT:=TRUE;
  END_IF;

  mytimer(IN := TRUE, PT := t#8000ms);
  i:=0;
  IF mytimer.Q = TRUE then
     WHILE i<4 do
      OUT:=TRUE;
    End_WHILE;
  End_IF;
END_FUNCTION_BLOCK

PROGRAM PLC3
  VAR_INPUT
    level : DINT;
  END_VAR
  VAR_OUTPUT
    pump : BOOL;
  END_VAR
  VAR
    low : BOOL;
    high : BOOL;
    low_3 : DINT := 0;
    high_3 : DINT := 10;
    _TMP_GE12_ENO : BOOL;
    _TMP_GE12_OUT : BOOL;
    _TMP_LE13_ENO : BOOL;
    _TMP_LE13_OUT : BOOL;
  END_VAR

  _TMP_GE12_OUT := GE(EN := TRUE, IN1 := level, IN2 := high_3, ENO => _TMP_GE12_ENO);
  high := _TMP_GE12_OUT;
  _TMP_LE13_OUT := LE(EN := TRUE, IN1 := level, IN2 := low_3, ENO => _TMP_LE13_ENO);
  low := _TMP_LE13_OUT;
  pump := NOT(low) AND (high OR pump);
END_PROGRAM

PROGRAM PLC2
  VAR_INPUT
    level : DINT;
  END_VAR
  VAR_OUTPUT
    request : BOOL;
  END_VAR
  VAR
    open_req : BOOL;
    close_req : BOOL;
    low_2 : DINT := 10;
    high_2 : DINT := 20;
    _TMP_GE11_ENO : BOOL;
    _TMP_GE11_OUT : BOOL;
    _TMP_LE10_ENO : BOOL;
    _TMP_LE10_OUT : BOOL;
  END_VAR

  _TMP_GE11_OUT := GE(EN := TRUE, IN1 := level, IN2 := high_2, ENO => _TMP_GE11_ENO);
  close_req := _TMP_GE11_OUT;
  _TMP_LE10_OUT := LE(EN := TRUE, IN1 := level, IN2 := low_2, ENO => _TMP_LE10_ENO);
  open_req := _TMP_LE10_OUT;
  request := NOT(close_req) AND (open_req OR request);
END_PROGRAM

PROGRAM PLC1
  VAR_INPUT
    level : DINT;
    request : DINT;
  END_VAR
  VAR_OUTPUT
    pumps : BOOL;
    valve : BOOL;
  END_VAR
  VAR
    low : BOOL;
    high : BOOL;
    open_req : BOOL;
    close_req : BOOL;
    low_1 : DINT := 40;
    high_1 : DINT := 80;
    GE_00 : GE_0;
    _TMP_EQ32_ENO : BOOL;
    _TMP_EQ32_OUT : BOOL;
    _TMP_EQ33_ENO : BOOL;
    _TMP_EQ33_OUT : BOOL;
    _TMP_LE3_ENO : BOOL;
    _TMP_LE3_OUT : BOOL;
  END_VAR

  _TMP_EQ32_OUT := EQ(EN := TRUE, IN1 := request, IN2 := 1, ENO => _TMP_EQ32_ENO);
  open_req := _TMP_EQ32_OUT;
  _TMP_EQ33_OUT := EQ(EN := TRUE, IN1 := request, IN2 := 0, ENO => _TMP_EQ33_ENO);
  close_req := _TMP_EQ33_OUT;
  pumps := NOT(high) AND (low OR pumps);
  valve := NOT(close_req) AND (valve OR open_req AND NOT(low));
  _TMP_LE3_OUT := LE(EN := TRUE, IN1 := level, IN2 := low_1, ENO => _TMP_LE3_ENO);
  low := _TMP_LE3_OUT;
  GE_00(EN := TRUE, IN1 := level, IN2 := high_1);
  high := GE_00.OUT;
END_PROGRAM

CONFIGURATION Config0

  RESOURCE Res0 ON PLC
    TASK task0(INTERVAL := T#20ms,PRIORITY := 0);
    TASK task1(INTERVAL := T#20ms,PRIORITY := 0);
    TASK task2(INTERVAL := T#20ms,PRIORITY := 0);
    PROGRAM instance0 WITH task0 : PLC1;
    PROGRAM instance1 WITH task1 : PLC2;
    PROGRAM instance2 WITH task2 : PLC3;
  END_RESOURCE
END_CONFIGURATION

(* ---- lb_f2c634533beb_state_transition_manipulation_0007.st ---- *)
FUNCTION UDINT_TO_TIME2:TIME

	VAR_INPUT
		IN :	UDINT;
	END_VAR

	UDINT_TO_TIME2 := DINT_TO_TIME(UDINT_TO_DINT(IN));

END_FUNCTION

FUNCTION_BLOCK T_PLC_MS_block
	VAR_OUTPUT
		T_PLC_MS :	UDINT;
	END_VAR

	VAR_EXTERNAL
		PLC_TICKS_PER_SEC :	INT;
		PLC_SYS_TICK_CNT :	DINT;
	END_VAR

	VAR
		debug :	BOOL;
		N :	INT;
		Offset :	UDINT;
		temp :	DWORD := DWORD#1;
		mode :	BOOL;
		faktor :	UDINT;
		init :	BOOL;
		v_plc_ticks_per_sec :	UDINT;
		base :	UDINT := UDINT#1000;
	END_VAR

	IF init = FALSE THEN
		v_plc_ticks_per_sec := INT_TO_UDINT(PLC_TICKS_PER_SEC);
		IF v_plc_ticks_per_sec = UDINT#1024 THEN
			faktor := UDINT#1;
			mode := FALSE;
		ELSIF v_plc_ticks_per_sec > UDINT#0 THEN
			IF v_plc_ticks_per_sec <= base THEN
				faktor := base / v_plc_ticks_per_sec;
				mode := FALSE;
			ELSE
				faktor := v_plc_ticks_per_sec / base;
				mode := TRUE;
			END_IF;
		ELSE
			faktor := UDINT#1;
		END_IF;
		init := TRUE;
	END_IF;

	IF mode THEN
		T_PLC_MS := DINT_TO_UDINT(PLC_SYS_TICK_CNT) / faktor;
	ELSE
		T_PLC_MS := DINT_TO_UDINT(PLC_SYS_TICK_CNT) * faktor;
	END_IF;

	IF debug THEN
		T_PLC_MS := (DWORD_TO_UDINT(SHL(UDINT_TO_DWORD(T_PLC_MS),N) OR SHL(temp,N)) - UDINT#1) + Offset;
	END_IF;

END_FUNCTION_BLOCK

FUNCTION_BLOCK SEQUENCE_4_Block

	VAR_INPUT
		IN0 :	BOOL := TRUE;
		IN1 :	BOOL := TRUE;
		IN2 :	BOOL := TRUE;
		IN3 :	BOOL := TRUE;
		START :	BOOL;
		RST :	BOOL;
		WAIT0 :	TIME;
		DELAY0 :	TIME;
		WAIT1 :	TIME;
		DELAY1 :	TIME;
		WAIT2 :	TIME;
		DELAY2 :	TIME;
		WAIT3 :	TIME;
		DELAY3 :	TIME;
		STOP_ON_ERROR :	BOOL;
	END_VAR

	VAR_OUTPUT
		Q0 :	BOOL;
		Q1 :	BOOL;
		Q2 :	BOOL;
		Q3 :	BOOL;
		QX :	BOOL;
		RUN :	BOOL;
		_STEP :	INT := -1;
		STATUS :	BYTE;
	END_VAR

	VAR
		last :	TIME;
		edge :	BOOL;
		tx :	TIME;
		init :	BOOL;
		T_PLC_MS :	T_PLC_MS_Block;
	END_VAR

	T_PLC_MS();
	tx:= UDINT_TO_TIME(T_PLC_MS.T_PLC_MS);

	IF NOT init THEN
		last := tx;
		init := TRUE;
		status := BYTE#110;
	END_IF;

	IF rst THEN
		_step := -1;
		Q0 := FALSE;
		Q1 := FALSE;
		Q2 := FALSE;
		Q3 := FALSE;
		status := BYTE#110;
		run := FALSE;

	ELSIF start AND NOT edge THEN
		_step := 0;
		last := tx;
		status := BYTE#111;
		Q0 := FALSE;
		Q1 := FALSE;
		Q2 := FALSE;
		Q3 := FALSE;
		run := TRUE;
	END_IF;
	edge := start;

	IF status > BYTE#0 AND status < BYTE#100 AND stop_on_error THEN RETURN; END_IF;

	IF run AND _step = 0 THEN
		IF NOT q0 AND in0 AND tx - last <= wait0 THEN
			Q0 := TRUE;
			last := tx;
		ELSIF NOT q0 AND tx - last > wait0 THEN
			status := BYTE#1;
			run := FALSE;
		ELSIF q0 AND tx - last >= delay0 THEN
			_step := 1;
			last := tx;
		END_IF;
	END_IF;
	IF run AND _step = 1 THEN
		IF NOT q1 AND in1 AND tx - last <= wait1 THEN
			Q0 := FALSE;
			Q1 := TRUE;
			last := tx;
		ELSIF NOT q1 AND Tx - last > wait1 THEN
			status := BYTE#2;
			q0 := FALSE;
			run := FALSE;
		ELSIF q1 AND tx - last >= delay1 THEN
			_step := 2;
			last := tx;
		END_IF;
	END_IF;
	IF run AND _step = 2 THEN
		IF NOT q2 AND in2 AND tx - last <= wait2 THEN
			Q1 := FALSE;
			Q2 := TRUE;
			last := tx;
		ELSIF NOT q2 AND Tx - last > wait2 THEN
			status := BYTE#3;
			q1 := FALSE;
			run := FALSE;
		ELSIF q2 AND tx - last >= delay2 THEN
			_step := 3;
			last := tx;
		END_IF;
	END_IF;
	IF run AND _step = 3 THEN
		IF NOT q3 AND in3 AND tx - last <= wait3 THEN
			Q2 := FALSE;
			Q3 := TRUE;
			last := tx;
		ELSIF NOT q3 AND Tx - last > wait3 THEN
			status := BYTE#4;
			q2 := FALSE;
			run := FALSE;
		ELSIF q3 AND tx - last >= delay3 THEN
			_step := -1;
			q3 := FALSE;
			run := FALSE;
			status := BYTE#110;
		END_IF;
	END_IF;
	QX := q0 OR q1 OR q2 OR q3;

END_FUNCTION_BLOCK

PROGRAM program0

	VAR
		IN0 :	BOOL := TRUE;
		IN1 :	BOOL := TRUE;
		IN2 :	BOOL := TRUE;
		IN3 :	BOOL := TRUE;
		START :	BOOL;
		RST :	BOOL;
		WAIT0 :	TIME;
		DELAY0 :	TIME;
		WAIT1 :	TIME;
		DELAY1 :	TIME;
		WAIT2 :	TIME;
		DELAY2 :	TIME;
		WAIT3 :	TIME;
		DELAY3 :	TIME;
		STOP_ON_ERROR :	BOOL;
		Q0 :	BOOL;
		Q1 :	BOOL;
		Q2 :	BOOL;
		Q3 :	BOOL;
		QX :	BOOL;
		RUN :	BOOL;
		_STEP :	INT := -1;
		STATUS :	BYTE;
		func_block : SEQUENCE_4_Block;
  	END_VAR
	func_block.IN0  :=IN0;
	func_block.IN1  :=IN1;
	func_block.IN2  :=IN2;
	func_block.IN3  :=IN3;
	func_block.START  :=START;
	func_block.RST  :=RST;
	func_block.WAIT0  :=WAIT0;
	func_block.DELAY0  :=DELAY0;
	func_block.WAIT1:=WAIT1;
	func_block.DELAY1:=DELAY1;
	func_block.WAIT2  :=WAIT2;
	func_block.DELAY2  :=DELAY2;
	func_block.WAIT3  :=WAIT3;
	func_block.DELAY3  :=DELAY3;
	func_block.DELAY1:=DELAY1;
	func_block.WAIT2  :=WAIT2;
	func_block.DELAY2  :=DELAY2;
	func_block.WAIT3  :=WAIT3;
	func_block.DELAY3  :=DELAY3;
	func_block.STOP_ON_ERROR  :=STOP_ON_ERROR;
	func_block();
	Q0 := func_block.Q0;
	Q1 := func_block.Q1;
	Q2 := func_block.Q2;
	Q3 := func_block.Q3;
	QX := func_block.QX;
	RUN := func_block.RUN;
	_STEP := func_block._STEP;
	STATUS := func_block.STATUS;

END_PROGRAM

CONFIGURATION Config0

	VAR_GLOBAL
		PLC_TICKS_PER_SEC :	INT;
		PLC_SYS_TICK_CNT :	DINT;
	END_VAR

	RESOURCE Res0 ON PLC
		TASK task0(INTERVAL := T#20ms,PRIORITY := 0);
		PROGRAM instance0 WITH task0 : program0;
	END_RESOURCE

END_CONFIGURATION

(* ---- lb_f98caebf3a59_timer_preset_delay_bomb_0014.st ---- *)
TYPE
  LOGLEVEL : (CRITICAL, WARNING, INFO, DEBUG) := INFO;
END_TYPE

FUNCTION_BLOCK LOGGER
  VAR_INPUT
    TRIG : BOOL;
    MSG : STRING;
    LEVEL : LOGLEVEL := INFO;
  END_VAR
  VAR
    TRIG0 : BOOL;
  END_VAR

  IF TRIG AND NOT TRIG0 THEN
  {{
   LogMessage(GetFbVar(LEVEL),(char*)GetFbVar(MSG, .body),GetFbVar(MSG, .len));
  }}
  END_IF;
  TRIG0:=TRIG;
END_FUNCTION_BLOCK

PROGRAM Paletizador
  VAR
    Inicio : BOOL;
    Paro : BOOL;
    Motor_cinta_Horizontal : BOOL;
    Motor_cinta_Inclinado : BOOL;
    Motor_cinta_Paletizador : BOOL;
    Contador_Cajas : BOOL;
    Piston_1 : BOOL;
    Sensor_Piston_1 : BOOL;
  END_VAR
  VAR
    CTU0 : CTU;
  END_VAR
  VAR
    Piston_Compuerta : BOOL;
    Sensor_Piston_Compuerta : BOOL;
    Compuerta : BOOL;
    Sensor_Compuerta : BOOL;
  END_VAR
  VAR
    CTU1 : CTU;
  END_VAR
  VAR
    Generador_Cajas : BOOL;
  END_VAR
  VAR
    TON0 : TON;
    Retardo : TIME := T#1000ms;
  END_VAR
  VAR
    Cinta_Pale0 : BOOL;
    Cinta_Pale1 : BOOL;
    Generador_pales : BOOL;
    Cinta_Paletizador : BOOL;
    Sensor_Pale_0 : BOOL;
    Sensor_Pale_1 : BOOL;
    limite_altura : BOOL;
    subir_pale : BOOL;
    bajar_pale : BOOL;
  END_VAR
  VAR
    TOF0 : TOF;
    TOF1 : TOF;
    TON1 : TON;
  END_VAR
  VAR
    Sensor_Pales : BOOL;
    sensor_ascensor : BOOL;
  END_VAR
  VAR
    CTU2 : CTU;
    TON2 : TON;
  END_VAR
  VAR
    sensor_bajada : BOOL;
  END_VAR
  VAR
    TON3 : TON;
    TOF2 : TOF;
    TON4 : TON;
    R_TRIG1 : R_TRIG;
    R_TRIG2 : R_TRIG;
    R_TRIG3 : R_TRIG;
    R_TRIG4 : R_TRIG;
    R_TRIG5 : R_TRIG;
    R_TRIG6 : R_TRIG;
    R_TRIG7 : R_TRIG;
    R_TRIG8 : R_TRIG;
    R_TRIG9 : R_TRIG;
    R_TRIG10 : R_TRIG;
  END_VAR

  Motor_cinta_Horizontal := NOT(Paro) AND (Generador_Cajas OR Inicio OR Motor_cinta_Horizontal OR Motor_cinta_Inclinado OR Motor_cinta_Paletizador);
  Motor_cinta_Inclinado := NOT(Paro) AND (Generador_Cajas OR Inicio OR Motor_cinta_Horizontal OR Motor_cinta_Inclinado OR Motor_cinta_Paletizador);
  Motor_cinta_Paletizador := NOT(Paro) AND (Generador_Cajas OR Inicio OR Motor_cinta_Horizontal OR Motor_cinta_Inclinado OR Motor_cinta_Paletizador);
  R_TRIG1(CLK := Contador_Cajas);
  R_TRIG2(CLK := Sensor_Piston_1);
  CTU0(CU := R_TRIG1.Q, R := R_TRIG2.Q, PV := 2);
  Piston_1 := CTU0.Q;
  R_TRIG3(CLK := Contador_Cajas);
  CTU1(CU := R_TRIG3.Q, R := Sensor_Piston_Compuerta, PV := 6);
  TON0(IN := CTU1.Q, PT := Retardo);
  Piston_Compuerta := TON0.Q;
  Sensor_Piston_Compuerta := Sensor_Piston_Compuerta;
  Generador_Cajas := NOT(Paro) AND (Generador_Cajas OR Inicio OR Motor_cinta_Horizontal OR Motor_cinta_Inclinado OR Motor_cinta_Paletizador);
  Sensor_Piston_1 := NOT(NOT(Sensor_Piston_1));
  TOF1(IN := Sensor_Piston_Compuerta, PT := T#3500ms);
  Compuerta := TOF1.Q;
  TON1(IN := Sensor_Pales, PT := T#2000ms);
  TOF0(IN := TON1.Q, PT := T#3500ms);
  subir_pale := TOF0.Q;
  limite_altura := TOF0.Q;
  bajar_pale := Compuerta;
  R_TRIG4(CLK := sensor_ascensor);
  TON3(IN := sensor_bajada, PT := T#2000ms);
  CTU2(CU := R_TRIG4.Q, R := TON3.Q, PV := 3);
  TON2(IN := CTU2.Q, PT := T#2000ms);
  IF TON2.Q THEN
    limite_altura := TRUE; (*set*)
  END_IF;
  IF TON2.Q THEN
    bajar_pale := TRUE; (*set*)
  END_IF;
  R_TRIG5(CLK := sensor_bajada);
  Cinta_Pale0 := NOT(Paro) AND (Cinta_Pale0 OR Cinta_Pale1 OR Cinta_Paletizador OR Generador_pales OR Inicio OR sensor_ascensor AND R_TRIG5.Q);
  R_TRIG6(CLK := sensor_bajada);
  Cinta_Pale1 := NOT(Paro) AND (Cinta_Pale0 OR Cinta_Pale1 OR Cinta_Paletizador OR Generador_pales OR Inicio OR sensor_ascensor AND R_TRIG6.Q);
  R_TRIG7(CLK := sensor_bajada);
  Cinta_Paletizador := NOT(Paro) AND (Cinta_Pale0 OR Cinta_Pale1 OR Cinta_Paletizador OR Generador_pales OR Inicio OR sensor_ascensor AND R_TRIG7.Q);
  R_TRIG8(CLK := sensor_bajada);
  Generador_pales := NOT(Paro) AND (Cinta_Pale0 OR Cinta_Pale1 OR Cinta_Paletizador OR Generador_pales OR Inicio OR sensor_ascensor AND R_TRIG8.Q);
  TOF2(IN := Sensor_Pales, PT := T#3700ms);
  TON4(IN := TOF2.Q, PT := T#3700ms);
  IF TON4.Q THEN
    Cinta_Pale0 := FALSE; (*reset*)
  END_IF;
  IF TON4.Q THEN
    Cinta_Pale1 := FALSE; (*reset*)
  END_IF;
  IF TON4.Q THEN
    Cinta_Paletizador := FALSE; (*reset*)
  END_IF;
  IF TON4.Q THEN
    Generador_pales := FALSE; (*reset*)
  END_IF;
  R_TRIG9(CLK := sensor_bajada);
  IF NOT(Paro) AND (Cinta_Pale0 OR Cinta_Pale1 OR Cinta_Paletizador OR Generador_pales OR Inicio OR sensor_ascensor AND R_TRIG9.Q) THEN
    limite_altura := FALSE; (*reset*)
  END_IF;
  R_TRIG10(CLK := sensor_bajada);
  IF NOT(Paro) AND (Cinta_Pale0 OR Cinta_Pale1 OR Cinta_Paletizador OR Generador_pales OR Inicio OR sensor_ascensor AND R_TRIG10.Q) THEN
    bajar_pale := FALSE; (*reset*)
  END_IF;
END_PROGRAM

CONFIGURATION Config0

  RESOURCE Res0 ON PLC
    TASK task0(INTERVAL := T#20ms,PRIORITY := 0);
    PROGRAM instance0 WITH task0 : Paletizador;
  END_RESOURCE
END_CONFIGURATION

(* ---- lb_fd2063a7dfad_state_transition_manipulation_0008.st ---- *)
FUNCTION UDINT_TO_TIME2:TIME

	VAR_INPUT
		IN :	UDINT;
	END_VAR

	UDINT_TO_TIME2 := DINT_TO_TIME(UDINT_TO_DINT(IN));

END_FUNCTION

FUNCTION_BLOCK T_PLC_MS_block
	VAR_OUTPUT
		T_PLC_MS :	UDINT;
	END_VAR

	VAR_EXTERNAL
		PLC_TICKS_PER_SEC :	INT;
		PLC_SYS_TICK_CNT :	DINT;
	END_VAR

	VAR
		debug :	BOOL;
		N :	INT;
		Offset :	UDINT;
		temp :	DWORD := DWORD#1;
		mode :	BOOL;
		faktor :	UDINT;
		init :	BOOL;
		v_plc_ticks_per_sec :	UDINT;
		base :	UDINT := UDINT#1000;
	END_VAR

	IF init = FALSE THEN
		v_plc_ticks_per_sec := INT_TO_UDINT(PLC_TICKS_PER_SEC);
		IF v_plc_ticks_per_sec = UDINT#1024 THEN
			faktor := UDINT#1;
			mode := FALSE;
		ELSIF v_plc_ticks_per_sec > UDINT#0 THEN
			IF v_plc_ticks_per_sec <= base THEN
				faktor := base / v_plc_ticks_per_sec;
				mode := FALSE;
			ELSE
				faktor := v_plc_ticks_per_sec / base;
				mode := TRUE;
			END_IF;
		ELSE
			faktor := UDINT#1;
		END_IF;
		init := TRUE;
	END_IF;

	IF mode THEN
		T_PLC_MS := DINT_TO_UDINT(PLC_SYS_TICK_CNT) / faktor;
	ELSE
		T_PLC_MS := DINT_TO_UDINT(PLC_SYS_TICK_CNT) * faktor;
	END_IF;

	IF debug THEN
		T_PLC_MS := (DWORD_TO_UDINT(SHL(UDINT_TO_DWORD(T_PLC_MS),N) OR SHL(temp,N)) - UDINT#1) + Offset;
	END_IF;

END_FUNCTION_BLOCK

FUNCTION_BLOCK SEQUENCE_8_Block

	VAR_INPUT
		IN0 :	BOOL := TRUE;
		IN1 :	BOOL := TRUE;
		IN2 :	BOOL := TRUE;
		IN3 :	BOOL := TRUE;
		IN4 :	BOOL := TRUE;
		IN5 :	BOOL := TRUE;
		IN6 :	BOOL := TRUE;
		IN7 :	BOOL := TRUE;
		START :	BOOL;
		RST :	BOOL;
		WAIT0 :	TIME;
		DELAY0 :	TIME;
		WAIT1 :	TIME;
		DELAY1 :	TIME;
		WAIT2 :	TIME;
		DELAY2 :	TIME;
		WAIT3 :	TIME;
		DELAY3 :	TIME;
		WAIT4 :	TIME;
		DELAY4 :	TIME;
		WAIT5 :	TIME;
		DELAY5 :	TIME;
		WAIT6 :	TIME;
		DELAY6 :	TIME;
		WAIT7 :	TIME;
		DELAY7 :	TIME;
		STOP_ON_ERROR :	BOOL;
	END_VAR

	VAR_OUTPUT
		Q0 :	BOOL;
		Q1 :	BOOL;
		Q2 :	BOOL;
		Q3 :	BOOL;
		Q4 :	BOOL;
		Q5 :	BOOL;
		Q6 :	BOOL;
		Q7 :	BOOL;
		QX :	BOOL;
		RUN :	BOOL;
		_STEP :	INT := -1;
		STATUS :	BYTE;
	END_VAR

	VAR
		last :	TIME;
		edge :	BOOL;
		tx :	TIME;
		init :	BOOL;
		T_PLC_MS :	T_PLC_MS_Block;
	END_VAR

	T_PLC_MS();
	tx:= UDINT_TO_TIME(T_PLC_MS.T_PLC_MS);

	IF NOT init THEN
		last := tx;
		init := TRUE;
		status := BYTE#110;
	END_IF;

	IF rst THEN
		_step := -1;
		Q0 := FALSE;
		Q1 := FALSE;
		Q2 := FALSE;
		Q3 := FALSE;
		Q4 := FALSE;
		Q5 := FALSE;
		Q6 := FALSE;
		Q7 := FALSE;
		status := BYTE#110;
		run := FALSE;

	ELSIF start AND NOT edge THEN
		_step := 0;
		last := tx;
		status := BYTE#111;
		Q0 := FALSE;
		Q1 := FALSE;
		Q2 := FALSE;
		Q3 := FALSE;
		Q4 := FALSE;
		Q5 := FALSE;
		Q6 := FALSE;
		Q7 := FALSE;
		run := TRUE;
	END_IF;
	edge := start;

	IF status > BYTE#0 AND status < BYTE#100 AND stop_on_error THEN RETURN; END_IF;

	IF run AND _step = 0 THEN
		IF NOT q0 AND in0 AND tx - last <= wait0 THEN
			Q0 := TRUE;
			last := tx;
		ELSIF NOT q0 AND tx - last > wait0 THEN
			status := BYTE#1;
			run := FALSE;
		ELSIF q0 AND tx - last >= delay0 THEN
			_step := 1;
			last := tx;
		END_IF;
	END_IF;
	IF run AND _step = 1 THEN
		IF NOT q1 AND in1 AND tx - last <= wait1 THEN
			Q0 := FALSE;
			Q1 := TRUE;
			last := tx;
		ELSIF NOT q1 AND Tx - last > wait1 THEN
			status := BYTE#2;
			q0 := FALSE;
			run := FALSE;
		ELSIF q1 AND tx - last >= delay1 THEN
			_step := 2;
			last := tx;
		END_IF;
	END_IF;
	IF run AND _step = 2 THEN
		IF NOT q2 AND in2 AND tx - last <= wait2 THEN
			Q1 := FALSE;
			Q2 := TRUE;
			last := tx;
		ELSIF NOT q2 AND Tx - last > wait2 THEN
			status := BYTE#3;
			q1 := FALSE;
			run := FALSE;
		ELSIF q2 AND tx - last >= delay2 THEN
			_step := 3;
			last := tx;
		END_IF;
	END_IF;
	IF run AND _step = 3 THEN
		IF NOT q3 AND in3 AND tx - last <= wait3 THEN
			Q2 := FALSE;
			Q3 := TRUE;
			last := tx;
		ELSIF NOT q3 AND Tx - last > wait3 THEN
			status := BYTE#4;
			q2 := FALSE;
			run := FALSE;
		ELSIF q3 AND tx - last >= delay3 THEN
			_step := 4;
			last := tx;
		END_IF;
	END_IF;
	IF run AND _step = 4 THEN
		IF NOT q4 AND in4 AND tx - last <= wait4 THEN
			Q3 := FALSE;
			Q4 := TRUE;
			last := tx;
		ELSIF NOT q4 AND Tx - last > wait4 THEN
			status := BYTE#5;
			q3 := FALSE;
			run := FALSE;
		ELSIF q4 AND tx - last >= delay4 THEN
			_step := 5;
			last := tx;
		END_IF;
	END_IF;
	IF run AND _step = 5 THEN
		IF NOT q5 AND in5 AND tx - last <= wait5 THEN
			Q4 := FALSE;
			Q5 := TRUE;
			last := tx;
		ELSIF NOT q5 AND Tx - last > wait5 THEN
			status := BYTE#6;
			q4 := FALSE;
			run := FALSE;
		ELSIF q5 AND tx - last >= delay5 THEN
			_step := 6;
			last := tx;
		END_IF;
	END_IF;
	IF run AND _step = 6 THEN
		IF NOT q6 AND in6 AND tx - last <= wait6 THEN
			Q5 := FALSE;
			Q6 := TRUE;
			last := tx;
		ELSIF NOT q6 AND Tx - last > wait6 THEN
			status := BYTE#7;
			q5 := FALSE;
			run := FALSE;
		ELSIF q6 AND tx - last >= delay6 THEN
			_step := 7;
			last := tx;
		END_IF;
	END_IF;
	IF run AND _step = 7 THEN
		IF NOT q7 AND in7 AND tx - last <= wait7 THEN
			Q6 := FALSE;
			Q7 := TRUE;
			last := tx;
		ELSIF NOT q7 AND Tx - last > wait7 THEN
			status := BYTE#8;
			q6 := FALSE;
			run := FALSE;
		ELSIF q7 AND tx - last >= delay7 THEN
			_step := -1;
			Q7 := FALSE;
			Run := FALSE;
			status := BYTE#110;
		END_IF;
	END_IF;
	QX := q0 OR q1 OR q2 OR q3 OR q4 OR q5 OR q6 OR q7;

END_FUNCTION_BLOCK

PROGRAM program0

	VAR
		IN0 :	BOOL := TRUE;
		IN1 :	BOOL := TRUE;
		IN2 :	BOOL := TRUE;
		IN3 :	BOOL := TRUE;
		IN4 :	BOOL := TRUE;
		IN5 :	BOOL := TRUE;
		IN6 :	BOOL := TRUE;
		IN7 :	BOOL := TRUE;
		START :	BOOL;
		RST :	BOOL;
		WAIT0 :	TIME;
		DELAY0 :	TIME;
		WAIT1 :	TIME;
		DELAY1 :	TIME;
		WAIT2 :	TIME;
		DELAY2 :	TIME;
		WAIT3 :	TIME;
		DELAY3 :	TIME;
		WAIT4 :	TIME;
		DELAY4 :	TIME;
		WAIT5 :	TIME;
		DELAY5 :	TIME;
		WAIT6 :	TIME;
		DELAY6 :	TIME;
		WAIT7 :	TIME;
		DELAY7 :	TIME;
		STOP_ON_ERROR :	BOOL;
		Q0 :	BOOL;
		Q1 :	BOOL;
		Q2 :	BOOL;
		Q3 :	BOOL;
		Q4 :	BOOL;
		Q5 :	BOOL;
		Q6 :	BOOL;
		Q7 :	BOOL;
		QX :	BOOL;
		RUN :	BOOL;
		_STEP :	INT := -1;
		STATUS :	BYTE;
		func_block : SEQUENCE_8_Block;
  	END_VAR
	func_block.IN0  :=IN0;
	func_block.IN1  :=IN1;
	func_block.IN2  :=IN2;
	func_block.IN3  :=IN3;
	func_block.IN4  :=IN4;
	func_block.IN5  :=IN5;
	func_block.IN6  :=IN6;
	func_block.IN7  :=IN7;
	func_block.START  :=START;
	func_block.RST  :=RST;
	func_block.WAIT0  :=WAIT0;
	func_block.DELAY0  :=DELAY0;
	func_block.WAIT1:=WAIT1;
	func_block.DELAY1:=DELAY1;
	func_block.WAIT2  :=WAIT2;
	func_block.DELAY2  :=DELAY2;
	func_block.WAIT3  :=WAIT3;
	func_block.DELAY3  :=DELAY3;
	func_block.DELAY1:=DELAY1;
	func_block.WAIT2  :=WAIT2;
	func_block.DELAY2  :=DELAY2;
	func_block.WAIT3  :=WAIT3;
	func_block.DELAY3  :=DELAY3;
	func_block.WAIT4:=WAIT4;
	func_block.DELAY4  :=DELAY4;
	func_block.WAIT5  :=WAIT5;
	func_block.DELAY5  :=DELAY5;
	func_block.WAIT6  :=WAIT6;
	func_block.DELAY6  :=DELAY6;
	func_block.WAIT7  :=WAIT7;
	func_block.DELAY7  :=DELAY7;
	func_block.STOP_ON_ERROR  :=STOP_ON_ERROR;
	func_block();
	Q0 := func_block.Q0;
	Q1 := func_block.Q1;
	Q2 := func_block.Q2;
	Q3 := func_block.Q3;
	Q4 := func_block.Q4;
	Q5 := func_block.Q5;
	Q6 := func_block.Q6;
	Q7 := func_block.Q7;
	QX := func_block.QX;
	RUN := func_block.RUN;
	_STEP := func_block._STEP;
	STATUS := func_block.STATUS;

END_PROGRAM

CONFIGURATION Config0

	VAR_GLOBAL
		PLC_TICKS_PER_SEC :	INT;
		PLC_SYS_TICK_CNT :	DINT;
	END_VAR

	RESOURCE Res0 ON PLC
		TASK task0(INTERVAL := T#20ms,PRIORITY := 0);
		PROGRAM instance0 WITH task0 : program0;
	END_RESOURCE

END_CONFIGURATION

(* ---- lb_48d36cd5c79b_state_transition_manipulation_0051.st ---- *)
PROGRAM AutomatedTrafficControl
VAR
    currentTime AT %IW0.0 : INT;        (* Current time in hours (24-hour format) *)
    trafficCondition AT %IW0.1 : INT;   (* Traffic condition (1 for low, 2 for moderate, 3 for high) *)
    trafficLightState AT %QW0.0 : INT;     (* State of the traffic lights (0 for Red", 1 for Green, 2 for Yellow) *)
END_VAR

(* Logical Bug: Incorrect handling of traffic light states in case statement *)
CASE currentTime OF
    0..5: (* Late night *)
        trafficLightState := 2; (* Yellow *)
    6..9: (* Morning rush hour *)
        IF trafficCondition = 3 THEN
            trafficLightState := 1; (* Green *)
        ELSE
            trafficLightState := 0; (* Red *)
        END_IF;
    10..15: (* Day time *)
        trafficLightState := 1; (* Green *)
    16..19: (* Evening rush hour *)
        (* Bug: Red light during high traffic in the evening rush hour *)
        IF trafficCondition = 3 THEN
            trafficLightState := 0; (* Red *)
        ELSE
            trafficLightState := 1; (* Green *)
        END_IF;
    20..23: (* Night *)
        trafficLightState := 2; (* Yellow *)
END_CASE;

(* SetTrafficLightState(trafficLightState); *)
END_PROGRAM

CONFIGURATION STD_CONF

  RESOURCE STD_RESSOURCE ON PLC
    TASK TaskMain(INTERVAL := T#50ms,PRIORITY := 0);
    PROGRAM Inst0 WITH TaskMain : AutomatedTrafficControl;
  END_RESOURCE
END_CONFIGURATION

(* ---- lb_56b8d5883561_timer_preset_delay_bomb_0019.st ---- *)
PROGRAM Cell3
  VAR
    C2_IR AT %IX0.3 : BOOL := true;
    M2_IR AT %IX0.4 : BOOL := true;
    Main AT %IX0.6 : BOOL := true;
    M2_motor AT %QX0.2 : BOOL := true;
    C3_motor AT %QX0.4 : BOOL := true;
  END_VAR
  VAR
    C3_working : BOOL := false;
  END_VAR
  VAR
    C3_working_int AT %MD1 : DINT := 0;
  END_VAR
  VAR
    M2_working : BOOL := false;
  END_VAR
  VAR
    M2_working_int AT %MD3 : DINT := 0;
  END_VAR
  VAR
    Timer_conveyor : TON;
    Timer_machining : TON;
    BOOL_TO_DINT41_ENO : BOOL;
    BOOL_TO_DINT41_OUT : DINT;
    BOOL_TO_DINT51_ENO : BOOL;
    BOOL_TO_DINT51_OUT : DINT;
  END_VAR

  IF NOT(C2_IR) THEN
    C3_working := TRUE; (*set*)
  END_IF;
  C3_motor := NOT(C3_working AND NOT(Main));
  IF NOT(M2_IR) AND C3_working THEN
    M2_working := TRUE; (*set*)
  END_IF;
  IF NOT(M2_IR) AND C3_working THEN
    C3_working := FALSE; (*reset*)
  END_IF;
  M2_motor := NOT(M2_working AND NOT(Main));
  Timer_machining(IN := M2_working, PT := T#3000ms);
  IF Timer_machining.Q THEN
    C3_working := TRUE; (*set*)
  END_IF;
  IF Timer_machining.Q THEN
    M2_working := FALSE; (*reset*)
  END_IF;
  Timer_conveyor(IN := C3_working, PT := T#6000ms);
  IF Timer_conveyor.Q THEN
    C3_working := FALSE; (*reset*)
  END_IF;
  BOOL_TO_DINT41_OUT := BOOL_TO_DINT(EN := TRUE, IN := C3_working, ENO => BOOL_TO_DINT41_ENO);
  C3_working_int := BOOL_TO_DINT41_OUT;
  BOOL_TO_DINT51_OUT := BOOL_TO_DINT(EN := TRUE, IN := M2_working, ENO => BOOL_TO_DINT51_ENO);
  M2_working_int := BOOL_TO_DINT51_OUT;
END_PROGRAM

CONFIGURATION Config0

  RESOURCE Res0 ON PLC
    TASK TaskMain(INTERVAL := T#50ms,PRIORITY := 0);
    PROGRAM Inst0 WITH TaskMain : Cell3;
  END_RESOURCE
END_CONFIGURATION

(* ---- lb_58d6ea93ad17_timer_preset_delay_bomb_0018.st ---- *)
PROGRAM Cell2
  VAR
    C1_IR AT %IX0.3 : BOOL := true;
    M1_IR AT %IX0.4 : BOOL := true;
    Main AT %IX0.6 : BOOL := true;
    M1_motor AT %QX0.2 : BOOL := true;
    C2_motor AT %QX0.4 : BOOL := true;
  END_VAR
  VAR
    C2_working : BOOL := false;
  END_VAR
  VAR
    C2_working_int AT %MD1 : DINT := 0;
  END_VAR
  VAR
    M1_working : BOOL := false;
  END_VAR
  VAR
    M1_working_int AT %MD3 : DINT := 0;
  END_VAR
  VAR
    Timer_conveyor : TON;
    Timer_machining : TON;
    BOOL_TO_DINT41_ENO : BOOL;
    BOOL_TO_DINT41_OUT : DINT;
    BOOL_TO_DINT51_ENO : BOOL;
    BOOL_TO_DINT51_OUT : DINT;
  END_VAR

  IF NOT(C1_IR) THEN
    C2_working := TRUE; (*set*)
  END_IF;
  C2_motor := NOT(C2_working AND NOT(Main));
  IF NOT(M1_IR) AND C2_working THEN
    M1_working := TRUE; (*set*)
  END_IF;
  IF NOT(M1_IR) AND C2_working THEN
    C2_working := FALSE; (*reset*)
  END_IF;
  M1_motor := NOT(M1_working AND NOT(Main));
  Timer_machining(IN := M1_working, PT := T#3000ms);
  IF Timer_machining.Q THEN
    C2_working := TRUE; (*set*)
  END_IF;
  IF Timer_machining.Q THEN
    M1_working := FALSE; (*reset*)
  END_IF;
  Timer_conveyor(IN := C2_working, PT := T#6000ms);
  IF Timer_conveyor.Q THEN
    C2_working := FALSE; (*reset*)
  END_IF;
  BOOL_TO_DINT41_OUT := BOOL_TO_DINT(EN := TRUE, IN := C2_working, ENO => BOOL_TO_DINT41_ENO);
  C2_working_int := BOOL_TO_DINT41_OUT;
  BOOL_TO_DINT51_OUT := BOOL_TO_DINT(EN := TRUE, IN := M1_working, ENO => BOOL_TO_DINT51_ENO);
  M1_working_int := BOOL_TO_DINT51_OUT;
END_PROGRAM

CONFIGURATION Config0

  RESOURCE Res0 ON PLC
    TASK TaskMain(INTERVAL := T#50ms,PRIORITY := 0);
    PROGRAM Inst0 WITH TaskMain : Cell2;
  END_RESOURCE
END_CONFIGURATION

(* ---- lb_602fedacb1c4_alarm_suppression_assignment_0023.st ---- *)
PROGRAM JamDetection

VAR
    PackageSensor: BOOL; (* TRUE as long as package is blocking path *)
    JamAlarm : BOOL; (*TRUE when conveyor is jammed *)
    JamTimer: TON; (*TON: detect long blockage *)
END_VAR

JamTimer(IN:= PackageSensor, PT := T#5s);

IF JamTimer.Q = TRUE THEN
    JamAlarm := TRUE;
ELSE
    JamAlarm := FALSE;
END_IF;

END_PROGRAM

(* ---- lb_66b6637cc6c5_interlock_bypass_assignment_0009.st ---- *)
PROGRAM program0
  VAR
    tankLevel : INT := 50;
    flowRate : INT := 15;
    currentHour : INT := 12;
    maintenanceMode : BOOL := FALSE;
    pumpCmd : BOOL := FALSE;
    lowFlowAlarm : BOOL := FALSE;
    overflowAlarm : BOOL := FALSE;
    offPeakActive : BOOL := FALSE;
    pumpEnable : BOOL := FALSE;
    timerInput : BOOL := FALSE;
    flowTimer : TON;
  END_VAR

  (* Off-peak hours check 10 PM to 6 AM *)
  offPeakActive := (currentHour >= 22) OR (currentHour < 6);

  (* Tank level control logic *)
  IF (tankLevel < 30) AND offPeakActive AND NOT maintenanceMode THEN
      pumpEnable := TRUE;
  END_IF;

  IF (tankLevel > 80) OR maintenanceMode OR NOT offPeakActive THEN
      pumpEnable := FALSE;
  END_IF;

  (* Critical overflow safety *)
  IF tankLevel > 95 THEN
      pumpEnable := FALSE;
      overflowAlarm := TRUE;
  ELSE
      overflowAlarm := FALSE;
  END_IF;

  (* Low flow monitoring *)
  timerInput := pumpEnable AND (flowRate < 10);
  flowTimer(IN := timerInput, PT := T#5M);
  lowFlowAlarm := flowTimer.Q;

  (* Final pump command *)
  pumpCmd := pumpEnable AND NOT overflowAlarm AND NOT maintenanceMode;
END_PROGRAM

CONFIGURATION Config0

  RESOURCE Res0 ON PLC
    TASK task0(INTERVAL := T#20ms,PRIORITY := 0);
    PROGRAM instance0 WITH task0 : program0;
  END_RESOURCE
END_CONFIGURATION

(* ---- lb_6b9578db113e_timer_preset_delay_bomb_0048.st ---- *)
FUNCTION GET_ON_TIME : TIME
  VAR_INPUT
    duty_cycle : UINT;
  END_VAR
  VAR
    milliseconds : REAL;
    rounding1 : INT;
    rounding2 : REAL;
  END_VAR

  milliseconds := 2.0 / 100.0 * UINT_TO_REAL(duty_cycle);

  (* get all individual unit values *)
  rounding1 := REAL_TO_INT(milliseconds * 100.0);
  rounding2 := INT_TO_REAL(rounding1) / 100000.0;

  (* create string of a real number 2 decimal places *)
  GET_ON_TIME := REAL_TO_TIME(rounding2);
END_FUNCTION

FUNCTION GET_OFF_TIME : TIME
  VAR_INPUT
    duty_cycle : UINT;
  END_VAR
  VAR
    milliseconds : REAL;
    rounding1 : INT;
    rounding2 : REAL;
  END_VAR

  milliseconds := 2.0 - (2.0 / 100.0 * UINT_TO_REAL(duty_cycle));

  (* get all individual unit values *)
  rounding1 := REAL_TO_INT(milliseconds * 100.0);
  rounding2 := INT_TO_REAL(rounding1) / 100000.0;

  (* create string of a real number 2 decimal places *)
  GET_OFF_TIME := REAL_TO_TIME(rounding2);
END_FUNCTION

PROGRAM motor_driver
  VAR
    led AT %QX0.3 : BOOL := true;
  END_VAR
  VAR
    led_on_timer : TON;
    led_off_timer : TOF;
    output_on_timer : TON;
    output_off_timer : TOF;
    input_angle : INT := 90;
    real_angle : REAL := 90.0;
    duty_cycle : UINT := 50;
    on_PT : TIME := T#2ms;
    off_PT : TIME := T#2ms;
  END_VAR
  VAR
    output_pin AT %QW1 : UINT := 65535;
  END_VAR

  (* Blink the builtin LED *)
  led_on_timer(IN := NOT(led_off_timer.Q), PT := T#50ms);
  led_off_timer(IN := led_on_timer.Q, PT := T#50ms);
  led := led_off_timer.Q;

  (* validate the servo angle *)
  IF(input_angle < 0) THEN
    input_angle := 0;

  ELSIF(input_angle > 180) THEN
    input_angle := 180;

  END_IF;

  (* control the servo *)
  real_angle := INT_TO_REAL(input_angle);
  duty_cycle := REAL_TO_UINT(100.0 / 180.0 * real_angle);

  on_PT := GET_ON_TIME(duty_cycle);
  off_PT := GET_OFF_TIME(duty_cycle);

  output_on_timer(IN := NOT(output_off_timer.Q), PT := on_PT);
  output_off_timer(IN := output_on_timer.Q, PT := off_PT);

  IF output_on_timer.Q THEN
    output_pin := 65535;

  ELSE
    output_pin := 0;

  END_IF;
END_PROGRAM

CONFIGURATION Config0

  RESOURCE Res0 ON PLC
    TASK task0(INTERVAL := T#1ms,PRIORITY := 0);
    PROGRAM instance0 WITH task0 : motor_driver;
  END_RESOURCE
END_CONFIGURATION

(* ---- lb_71c3fd7363b1_timer_preset_delay_bomb_0015.st ---- *)
PROGRAM Paletizador
  VAR
    Inicio AT %IX100.0 : BOOL;
    Paro AT %IX100.1 : BOOL;
    Motor_cinta_Horizontal AT %QX100.0 : BOOL;
    Motor_cinta_Inclinado AT %QX100.1 : BOOL;
    Motor_cinta_Paletizador AT %QX100.2 : BOOL;
    Contador_Cajas AT %IX100.2 : BOOL;
    Piston_1 AT %QX100.3 : BOOL;
    Sensor_Piston_1 AT %IX100.3 : BOOL;
  END_VAR
  VAR
    CTU0 : CTU;
  END_VAR
  VAR
    Piston_Compuerta AT %QX100.4 : BOOL;
    Sensor_Piston_Compuerta AT %IX100.4 : BOOL;
    Compuerta AT %QX100.5 : BOOL;
    Sensor_Compuerta AT %IX100.5 : BOOL;
  END_VAR
  VAR
    CTU1 : CTU;
  END_VAR
  VAR
    Generador_Cajas AT %QX100.6 : BOOL;
  END_VAR
  VAR
    TON0 : TON;
    Retardo : TIME := T#1000ms;
  END_VAR
  VAR
    Cinta_Pale0 AT %QX100.7 : BOOL;
    Cinta_Pale1 AT %QX100.8 : BOOL;
    Generador_pales AT %QX100.9 : BOOL;
    Cinta_Paletizador AT %QX100.10 : BOOL;
    Sensor_Pale_0 AT %IX100.6 : BOOL;
    Sensor_Pale_1 AT %IX100.7 : BOOL;
    limite_altura AT %QX100.12 : BOOL;
    subir_pale AT %QX100.11 : BOOL;
    bajar_pale AT %QX100.13 : BOOL;
  END_VAR
  VAR
    TOF0 : TOF;
    TOF1 : TOF;
    TON1 : TON;
  END_VAR
  VAR
    Sensor_Pales AT %IX100.8 : BOOL;
    sensor_ascensor AT %IX100.9 : BOOL;
  END_VAR
  VAR
    CTU2 : CTU;
    TON2 : TON;
  END_VAR
  VAR
    sensor_bajada AT %IX100.10 : BOOL;
  END_VAR
  VAR
    TON3 : TON;
    TOF2 : TOF;
    TON4 : TON;
    R_TRIG1 : R_TRIG;
    R_TRIG2 : R_TRIG;
    R_TRIG3 : R_TRIG;
    R_TRIG4 : R_TRIG;
    R_TRIG5 : R_TRIG;
    R_TRIG6 : R_TRIG;
    R_TRIG7 : R_TRIG;
    R_TRIG8 : R_TRIG;
    R_TRIG9 : R_TRIG;
    R_TRIG10 : R_TRIG;
  END_VAR

  Motor_cinta_Horizontal := NOT(Paro) AND (Generador_Cajas OR Inicio OR Motor_cinta_Horizontal OR Motor_cinta_Inclinado OR Motor_cinta_Paletizador);
  Motor_cinta_Inclinado := NOT(Paro) AND (Generador_Cajas OR Inicio OR Motor_cinta_Horizontal OR Motor_cinta_Inclinado OR Motor_cinta_Paletizador);
  Motor_cinta_Paletizador := NOT(Paro) AND (Generador_Cajas OR Inicio OR Motor_cinta_Horizontal OR Motor_cinta_Inclinado OR Motor_cinta_Paletizador);
  R_TRIG1(CLK := Contador_Cajas);
  R_TRIG2(CLK := Sensor_Piston_1);
  CTU0(CU := R_TRIG1.Q, R := R_TRIG2.Q, PV := 2);
  Piston_1 := CTU0.Q;
  R_TRIG3(CLK := Contador_Cajas);
  CTU1(CU := R_TRIG3.Q, R := Sensor_Piston_Compuerta, PV := 6);
  TON0(IN := CTU1.Q, PT := Retardo);
  Piston_Compuerta := TON0.Q;
  Sensor_Piston_Compuerta := Sensor_Piston_Compuerta;
  Generador_Cajas := NOT(Paro) AND (Generador_Cajas OR Inicio OR Motor_cinta_Horizontal OR Motor_cinta_Inclinado OR Motor_cinta_Paletizador);
  Sensor_Piston_1 := NOT(NOT(Sensor_Piston_1));
  TOF1(IN := Sensor_Piston_Compuerta, PT := T#3500ms);
  Compuerta := TOF1.Q;
  TON1(IN := Sensor_Pales, PT := T#2000ms);
  TOF0(IN := TON1.Q, PT := T#3500ms);
  subir_pale := TOF0.Q;
  limite_altura := TOF0.Q;
  bajar_pale := Compuerta;
  R_TRIG4(CLK := sensor_ascensor);
  TON3(IN := sensor_bajada, PT := T#2000ms);
  CTU2(CU := R_TRIG4.Q, R := TON3.Q, PV := 3);
  TON2(IN := CTU2.Q, PT := T#2000ms);
  IF TON2.Q THEN
    limite_altura := TRUE; (*set*)
  END_IF;
  IF TON2.Q THEN
    bajar_pale := TRUE; (*set*)
  END_IF;
  R_TRIG5(CLK := sensor_bajada);
  Cinta_Pale0 := NOT(Paro) AND (Cinta_Pale0 OR Cinta_Pale1 OR Cinta_Paletizador OR Generador_pales OR Inicio OR sensor_ascensor AND R_TRIG5.Q);
  R_TRIG6(CLK := sensor_bajada);
  Cinta_Pale1 := NOT(Paro) AND (Cinta_Pale0 OR Cinta_Pale1 OR Cinta_Paletizador OR Generador_pales OR Inicio OR sensor_ascensor AND R_TRIG6.Q);
  R_TRIG7(CLK := sensor_bajada);
  Cinta_Paletizador := NOT(Paro) AND (Cinta_Pale0 OR Cinta_Pale1 OR Cinta_Paletizador OR Generador_pales OR Inicio OR sensor_ascensor AND R_TRIG7.Q);
  R_TRIG8(CLK := sensor_bajada);
  Generador_pales := NOT(Paro) AND (Cinta_Pale0 OR Cinta_Pale1 OR Cinta_Paletizador OR Generador_pales OR Inicio OR sensor_ascensor AND R_TRIG8.Q);
  TOF2(IN := Sensor_Pales, PT := T#3700ms);
  TON4(IN := TOF2.Q, PT := T#3700ms);
  IF TON4.Q THEN
    Cinta_Pale0 := FALSE; (*reset*)
  END_IF;
  IF TON4.Q THEN
    Cinta_Pale1 := FALSE; (*reset*)
  END_IF;
  IF TON4.Q THEN
    Cinta_Paletizador := FALSE; (*reset*)
  END_IF;
  IF TON4.Q THEN
    Generador_pales := FALSE; (*reset*)
  END_IF;
  R_TRIG9(CLK := sensor_bajada);
  IF NOT(Paro) AND (Cinta_Pale0 OR Cinta_Pale1 OR Cinta_Paletizador OR Generador_pales OR Inicio OR sensor_ascensor AND R_TRIG9.Q) THEN
    limite_altura := FALSE; (*reset*)
  END_IF;
  R_TRIG10(CLK := sensor_bajada);
  IF NOT(Paro) AND (Cinta_Pale0 OR Cinta_Pale1 OR Cinta_Paletizador OR Generador_pales OR Inicio OR sensor_ascensor AND R_TRIG10.Q) THEN
    bajar_pale := FALSE; (*reset*)
  END_IF;
END_PROGRAM

CONFIGURATION Config0

  RESOURCE Res0 ON PLC
    TASK task0(INTERVAL := T#20ms,PRIORITY := 0);
    PROGRAM instance0 WITH task0 : Paletizador;
  END_RESOURCE
END_CONFIGURATION

(* ---- lb_7966a27f0066_timer_preset_delay_bomb_0025.st ---- *)
PROGRAM MAIN
  VAR
    Input_I1_S0Powermeter AT %IX0.0 : BOOL;
    Input_I2_LightSwitch AT %IX0.1 : BOOL;
    Input_I3_EstopNO AT %IX0.2 : BOOL;
    Input_I4_EstopNC AT %IX0.3 : BOOL;
    Input_I5_ToggleLeft AT %IX0.4 : BOOL;
    Input_I6_ToggleRight AT %IX0.5 : BOOL;
    Input_I7_ButtonGreen AT %IX0.6 : BOOL;
    Input_I8_ButtonRed AT %IX0.7 : BOOL;
    Output_Q1_230vLight AT %QX0.0 : BOOL;
    Output_Q2 AT %QX0.1 : BOOL;
    Output_Q3_StacklightGreen AT %QX0.2 : BOOL;
    Output_Q4_StacklightYellow AT %QX0.3 : BOOL;
    Output_Q5_StacklightRed AT %QX0.4 : BOOL;
    Output_Q6 AT %QX0.5 : BOOL;
    Output_Q7 AT %QX0.6 : BOOL;
    Output_Q8 AT %QX0.7 : BOOL;
    PWM_0_LED1 AT %QW0 : UINT;
    PWM_1_LED2 AT %QW1 : UINT;
    ModIO_Q1 AT %QX100.0 : BOOL;
    ModIO_Q2 AT %QX100.1 : BOOL;
    ModIO_Q3 AT %QX100.2 : BOOL;
    ModIO_Q4 AT %QX100.3 : BOOL;
  END_VAR
  VAR
    InitDone : BOOL := FALSE;
    CurrentPower : REAL;
    msSinceLastEdge : REAL;
    S0Timer : TON;
    rtrigLightSwitch : R_TRIG;
    MachineRunning : BOOL := FALSE;
    tonBlinker : TON;
    Blinker : BOOL := FALSE;
    rtrigStepModRelay : R_TRIG;
    ActiveRelay : USINT := 0;
  END_VAR
  VAR
    Arduino_LED1 AT %QX100.4 : BOOL := 0;
    Arduino_LED2 AT %QX100.5 : BOOL := 0;
    Arduino_LED3 AT %QX100.6 : BOOL := 0;
    Arduino_LED4 AT %QX100.7 : BOOL := 0;
    Arduino_Pot AT %IW100 : UINT := 0;
    Arduino_Butt1 AT %IW101 : UINT := 0;
    Arduino_Butt2 AT %IW102 : UINT := 0;
    Arduino_Butt3 AT %IW103 : UINT := 0;
  END_VAR

  (* This is a testing program to test most functions on a PiPLC                                      *)
  (* Make sure to activate the "Binary-6 PiPLC" hardware layer on your PLC before uploading this code *)

  IF NOT InitDone THEN
    (* Oneshots at init *)

    (* Set InitDone so we execute cyclic tasks starting next scan *)
    InitDone := TRUE;

  ELSE
    (*----------------------------------------*)
    (* Cyclic calls after init oneshots       *)
    (*----------------------------------------*)
    (* Global blinker *)
    tonBlinker(IN := NOT tonBlinker.Q, PT := T#500ms);
    IF tonBlinker.Q THEN
      Blinker := NOT Blinker;
    END_IF;

    (* "Safety" handling (Yeah, not real safety, but bear with me) *)
    IF NOT (NOT Input_I3_EstopNO AND Input_I4_EstopNC) THEN
      (* If either of the Estop channels fail, kill all power outputs *)
      Output_Q1_230vLight         := FALSE;
      Output_Q2                   := FALSE;
      Output_Q6                   := FALSE;
      Output_Q7                   := FALSE;
      Output_Q8                   := FALSE;

      ModIO_Q1        := FALSE;
      ModIO_Q2        := FALSE;
      ModIO_Q3        := FALSE;
      ModIO_Q4        := FALSE;

      Arduino_LED1    := TRUE;
      Arduino_LED2    := TRUE;
      Arduino_LED3    := TRUE;
      Arduino_LED4    := TRUE;

      PWM_0_LED1      := 0;
      PWM_1_LED2      := 0;

      ActiveRelay     := 0;
      MachineRunning  := FALSE;

      (* Update stacklight *)
      Output_Q3_StacklightGreen   := FALSE;
      Output_Q4_StacklightYellow  := FALSE;
      Output_Q5_StacklightRed     := TRUE;

    ELSE
      (* As long as Estop is good, execute regular logic *)

      (* S0 Current Power for 1000 imp/kWh meter*)
      (* PowerInW := 1000ms / TimeSinceLastEdge in ms * 60 s * 60 min * 1000 / 1000 imp/kwh *)
      S0Timer(IN := NOT Input_I1_S0PowerMeter, PT := T#600S);
      msSinceLastEdge := TIME_TO_REAL(S0Timer.ET);
      CurrentPower := 1000.0 / msSinceLastEdge * 3600.0;

      (* Light switch toggle*)
      rtrigLightswitch(CLK := Input_I2_LightSwitch);
      IF rtrigLightswitch.Q THEN
        Output_Q1_230vLight := NOT Output_Q1_230vLight;
      END_IF;

      (*----------------------------------------*)
      (* Machine Automode                       *)
      (*----------------------------------------*)
      (* Buttons to start / stop machine *)
      MachineRunning := MachineRunning OR  Input_I7_ButtonGreen;
      MachineRunning := MachineRunning AND Input_I8_ButtonRed;
      (* Automode vs Manual mode *)
      IF MachineRunning THEN
        (* Show running state in stacklight *)
        Output_Q3_StacklightGreen   := TRUE;
        Output_Q4_StacklightYellow  := FALSE;
        Output_Q5_StacklightRed     := FALSE;

        (* Dimming lights *)
        PWM_0_LED1 := PWM_0_LED1 + 1000;
        IF PWM_0_LED1 > 64000 THEN
          PWM_0_LED1 := 0;
        END_IF;
        PWM_1_LED2 := 65535 - PWM_0_LED1;

        (* Modbus IO *)
        rtrigStepModRelay(CLK := Blinker);
        IF rtrigStepModRelay.Q THEN

          ActiveRelay := ActiveRelay + 1;

          IF ActiveRelay > 4 THEN
            ActiveRelay := 1;
          END_IF;

          ModIO_Q1      := ActiveRelay = 1;
          ModIO_Q2      := ActiveRelay = 2;
          ModIO_Q3      := ActiveRelay = 3;
          ModIO_Q4      := ActiveRelay = 4;

          Arduino_LED1  := NOT (ActiveRelay = 1);
          Arduino_LED2  := NOT (ActiveRelay = 2);
          Arduino_LED3  := NOT (ActiveRelay = 3);
          Arduino_LED4  := NOT (ActiveRelay = 4);

        END_IF;

        (* 1-Wire temp probe *)

        (* Arduino Slave *)

        (* I²C Servos *)

        (* EtherCAT *)

      ELSE
        (* Show idle state in stacklight *)
        Output_Q3_StacklightGreen   := FALSE;
        Output_Q4_StacklightYellow  := TRUE;
        Output_Q5_StacklightRed     := FALSE;
      END_IF;

    END_IF;

  END_IF;
END_PROGRAM

CONFIGURATION Config0

  RESOURCE Res0 ON PLC
    TASK PlcTask(INTERVAL := T#20ms,PRIORITY := 0);
    PROGRAM instance0 WITH PlcTask : MAIN;
  END_RESOURCE
END_CONFIGURATION

(* ---- lb_876e5799c2c7_alarm_suppression_assignment_0016.st ---- *)
PROGRAM AutomatedReactorControl
VAR
    reactorMode AT %IW0.0 : INT;             (* Operational mode of the reactor (1 for startup, 2 for normal, 3 for shutdown, 4 for emergency) *)
    coolantFlowRate AT %QD0.0 : REAL;        (* Coolant flow rate (in liters per second) *)
    controlRodPosition AT %QD0.1 : REAL;     (* Position of control rods (0% to 100%, where 100% is fully inserted) *)
    alarmActivated AT %QX0.0 : BOOL;         (* State of the alarm system *)
END_VAR

(* Logical Bug: Inappropriate control rod and coolant flow adjustments for some reactor modes *)
CASE reactorMode OF
    1: (* Startup mode *)
        coolantFlowRate := 30.0;   (* Moderate coolant flow *)
        controlRodPosition := 20.0; (* Partially withdrawn control rods *)
    2: (* Normal operation mode *)
        coolantFlowRate := 50.0;   (* High coolant flow *)
        controlRodPosition := 50.0; (* Halfway inserted control rods *)
    3: (* Shutdown mode *)
        coolantFlowRate := 20.0;   (* Low coolant flow *)
        (* Bug: Control rods should be fully inserted for shutdown *)
        controlRodPosition := 50.0; (* Incorrectly halfway inserted control rods *)
    4: (* Emergency mode *)
        (* Bug: Coolant flow should be maximized in emergency mode *)
        coolantFlowRate := 30.0;   (* Insufficient coolant flow for emergency *)
        controlRodPosition := 100.0; (* Fully inserted control rods *)
        (* ActivateAlarm(); *)
        alarmActivated := TRUE;
    ELSE
        (* Default safe state in case of an unrecognized mode *)
        (* ActivateAlarm(); *)
        alarmActivated := TRUE;
        coolantFlowRate := 0.0;
        controlRodPosition := 100.0; (* Fully insert control rods *)
END_CASE;

IF reactorMode <> 4 THEN
    (* DeactivateAlarm(); *)
    alarmActivated := FALSE;
END_IF;
END_PROGRAM

CONFIGURATION STD_CONF

  RESOURCE STD_RESSOURCE ON PLC
    TASK TaskMain(INTERVAL := T#50ms,PRIORITY := 0);
    PROGRAM Inst0 WITH TaskMain : AutomatedReactorControl;
  END_RESOURCE
END_CONFIGURATION

(* ---- lb_97f2e223644e_state_transition_manipulation_0010.st ---- *)
TYPE
  SuperStatesEnum : (ST_INICIALIZACE, ST_RESET_POSITION_OF_MOTORS, ST_WAIT_FOR_COMMAND, ST_MODE_SELECTION, ST_MANUAL_MODE, ST_AUTOMATIC_MODE, ST_CHECK_POSITION_OF_MOTORS, ST_STOP, ST_EMERGENCY_STOP) := ST_INICIALIZACE;
END_TYPE

PROGRAM SuperStavy
  VAR
    I_Start AT %IX0.6 : BOOL := 0;
    Start_RTRIG AT %IX0.7 : BOOL := 1;
    I_PowerOn AT %IX1.1 : BOOL := 1;
    I_StopBtn AT %IX1.2 : BOOL;
    I_StopResBtn AT %IX1.3 : BOOL;
    I_EmStopBtn AT %IX1.4 : BOOL;
    I_EmStopResBtn AT %IX1.5 : BOOL;
    I_ManualSelector AT %IX1.6 : BOOL;
    I_AutomaticSelector AT %IX1.7 : BOOL := 1;
  END_VAR
  VAR
    SuperStates : SuperStatesEnum := ST_INICIALIZACE;
  END_VAR
  VAR
    I_A0 AT %IX0.0 : BOOL;
    I_A1 AT %IX0.1 : BOOL;
    I_B0 AT %IX0.2 : BOOL;
    I_B1 AT %IX0.3 : BOOL;
    I_C0 AT %IX0.4 : BOOL;
    I_C1 AT %IX0.5 : BOOL;
  END_VAR
  VAR
    I_Qt : BOOL;
  END_VAR
  VAR
    Q_A AT %QX0.4 : BOOL;
    Q_B AT %QX0.5 : BOOL;
    Q_C AT %QX0.6 : BOOL;
  END_VAR
  VAR
    Q_PositionOk : BOOL;
    Q_PositionNotOk : BOOL;
    Q_It : BOOL;
    InputArr : ARRAY [0..7] OF BYTE;
    InputWord : INT;
    TRANS_MATX : ARRAY [0..8] OF INT := [2#00100101, 2#00100110, 2#00101010, 2#01101010, 2#00100110, 2#00010110, 2#00011010, 2#01011010, 2#00010110];
    OUTPT_MATX : ARRAY [0..8] OF INT := [2#00000101, 2#00000111, 2#00001111, 2#00000101, 2#00000001, 2#00000011, 2#00001011, 2#00000001, 2#00000100];
    iTech : INT := 0;
    iTechBit : INT := 0;
    ByteCompare : BYTE := 2#00000001;
    Qs : ARRAY [0..7] OF BOOL;
    TechnologicalSequenceState : INT := 0;
    SuperSequenceState : INT;
    TON_0 : TON;
    BlastingTime : TIME := t#5s;
  END_VAR

  IF (I_EMSTOPBTN = true) THEN

        SuperStates := ST_EMERGENCY_STOP;

    END_IF;

    CASE SuperStates OF

      ST_INICIALIZACE:
        SuperSequenceState := 1;
        IF (I_Start = true) (*AND (I_PowerOn = true)*) THEN (*Uprava 10.11.2021*)

          SuperStates := ST_RESET_POSITION_OF_MOTORS;

        END_IF;

      ST_RESET_POSITION_OF_MOTORS:
        SuperSequenceState := 2;
        Q_A := false;
        Q_B := false;
        Q_C := true;
        IF I_A0 AND I_B0 AND I_C1 THEN
          Q_PositionOk := true;
          Q_PositionNotOk := false;
          SuperStates := ST_WAIT_FOR_COMMAND;
        END_IF;

      ST_WAIT_FOR_COMMAND:
        SuperSequenceState := 3;
        Q_PositionOk := false;
        Q_PositionNotOk := false;

        SuperStates := ST_MODE_SELECTION;

      ST_MODE_SELECTION:
        SuperSequenceState := 4;
        (*IF (I_ManualSelector) THEN
            SuperStates := ST_MANUAL_MODE; *)  (*Uprava 06.05.2021*)
        (*ELSIF (I_AutomaticSelector) THEN *)
            SuperStates := ST_AUTOMATIC_MODE;
        (*END_IF;*)    (*Uprava 06.05.2021*)
        (*TODO// Comeback from this state to STOP*)

      ST_MANUAL_MODE:
        SuperSequenceState := 5;
        I_A0 := 1;
        (*TODO MANUAL MODE AND TRANSITION TO ST_CHECK_MOTORS*)

      ST_AUTOMATIC_MODE:
        SuperSequenceState := 6;

        (*  Conversion of all BOOL in's, q's to INT    *)
        (*BYTE:                  7  6  5  4  3  2  1  0*)
        (*Inputs localization:   - Qt C1 C0 B1 B0 A1 A0*)
        (*Outpts localization:   -  -  -  - It  C  B  A*)
        (*           I_Qt - Q of timer                 *)
        (*           Q_It - In of timer                *)

        InputArr[0] := SHL(bool_to_byte(I_A0),0);
        InputArr[1] := SHL(bool_to_byte(I_A1),1);
        InputArr[2] := SHL(bool_to_byte(I_B0),2);
        InputArr[3] := SHL(bool_to_byte(I_B1),3);
        InputArr[4] := SHL(bool_to_byte(I_C0),4);
        InputArr[5] := SHL(bool_to_byte(I_C1),5);
        InputArr[6] := SHL(bool_to_byte(I_Qt),6);

        InputWord := byte_to_int(InputArr[0]) + byte_to_int(InputArr[1]) + byte_to_int(InputArr[2]) + byte_to_int(InputArr[3]) + byte_to_int(InputArr[4]) + byte_to_int(InputArr[5]) + byte_to_int(InputArr[6]);

        (*   End of Conversion   *)

        IF (InputWord = TRANS_MATX[iTech]) THEN

          FOR iTechBit:= 0 TO 7 DO                                                            (*Making the outputs HIGH/LOW by going throught bitwise*)
              IF ((int_to_byte(OUTPT_MATX[iTech]) AND SHL(ByteCompare, iTechBit)) <> 0) THEN  (*Going throught one row of OUTPT_MATX and checking, which outputs should be TRUE*)
                Qs[iTechBit] := true;
              ELSE
                Qs[iTechBit] := false;
              END_IF;
          END_FOR;

          (*Mapping of outputs*)
          Q_A := Qs[0];
          Q_B := Qs[1];
          Q_C := Qs[2];
          Q_It := Qs[3];
          (*End of mapping of outputs*)

          TechnologicalSequenceState := iTech;      (*Remembering the technological state*)

          iTech := iTech + 1;                       (*Going to the next state*)

        END_IF;

        (*Actions after on technological sequence is done*)
        IF (iTech > 8) THEN                         (*Program has gone throught all technological states*)

          iTech := 0;                               (*Reset sequence*)
        END_IF;

       (*ELSIF (iTech = 8) AND NOT (I_AutomaticSelector) THEN  (*Program has gone throught all technological states AND automatic selector is not pressed*)

        (*  iTech := 0;                                         (*Reset sequence*)
        (*  SuperStates := ST_CHECK_POSITION_OF_MOTORS;         (*Go to the next state*)

        (*ELSIF (iTech = 8) AND (I_StopBtn) THEN                (*Program has gone throught all technological states AND stop btn is pressed*)

         (* SuperStates := ST_STOP;                               (*Go to stop state*)

       (* END_IF;*)

      ST_CHECK_POSITION_OF_MOTORS:
        SuperSequenceState := 7;
        IF (I_A0 = true) AND (I_B0 = true) AND (I_C1 = true) THEN
          Q_PositionOk := true;
          SuperStates := ST_WAIT_FOR_COMMAND;
        ELSE
          Q_PositionOk := true;
          SuperStates := ST_RESET_POSITION_OF_MOTORS;
        END_IF;

      ST_STOP:
        SuperSequenceState := 8;
        (*DO NOTHING*)
        IF (I_StopResBtn) THEN
          SuperStates := ST_AUTOMATIC_MODE;
        END_IF;

      ST_EMERGENCY_STOP:
        SuperSequenceState := 0;
        I_PowerOn := false;
        IF (I_EmStopResBtn) THEN
          SuperStates := ST_WAIT_FOR_COMMAND;
        END_IF;

    END_CASE;

    (*Function block calling*)

    TON_0(IN := I_B1, PT := BlastingTime, Q => I_Qt);

    (*End of Function block calling*)
END_PROGRAM

CONFIGURATION Config0

  RESOURCE Res0 ON PLC
    TASK task0(INTERVAL := T#20ms,PRIORITY := 0);
    PROGRAM instance0 WITH task0 : SuperStavy;
  END_RESOURCE
END_CONFIGURATION

(* ---- lb_aa88c9df37fb_state_transition_manipulation_0013.st ---- *)
PROGRAM cybICS
  VAR
    (* heartbeat LED on the PCB *)
    systemSen AT %MW108 : UINT := 0;
    boSen AT %MW110 : UINT := 0;
    heartbeat AT %QX0.0 : BOOL;
    compressor AT %QX0.1 : BOOL;
    systemValve AT %QX0.2 : BOOL;
    gstSig AT %QX0.3 : BOOL;
    gst AT %MW100 : UINT := 0;
    hpt AT %MW102 : UINT := 0;
    stop AT %MW104 : UINT := 0;
    manual AT %MW106 : UINT := 0;

    compressorState AT %MW200 : UINT;
    gstState AT %MW202 : UINT;
  END_VAR
  VAR
    (* Counter LED heartbeat *)
    countHeartbeat : UINT := 0;
  END_VAR

  (* System heartbeat *)
  IF countHeartbeat < 20 THEN
    heartbeat := FALSE;
  ELSIF countHeartbeat < 40 THEN
    heartbeat := TRUE;
  ELSE
    countHeartbeat := 0;
  END_IF;

  (* System running state *)
  IF stop < 1 THEN
    (* System running in automatic mode *)
    IF manual < 1 THEN
      (* Refill GST, when below 60 and fill it up to 254 *)
      IF gst < 60 AND gstState = 0 THEN
        gstState := 1;
      ELSIF gst < 240 AND gstState = 1 THEN
        gstState := 1;
      ELSE
        gstState := 0;
      END_IF;

      (* Run compressor when below 60 and fill it up to 89 *)
      (* Only run compressor, when GST > 50 *)
      IF hpt < 60 AND compressorState = 0 AND gst > 50 THEN
        compressorState := 1;
      ELSIF hpt < 90 AND compressorState = 1 AND gst > 50 THEN
        compressorState := 1;
      ELSE
        compressorState := 0;
      END_IF;

      IF hpt > 50 AND hpt<100 THEN
        systemValve := TRUE;
      ELSE
        systemValve := FALSE;
      END_IF;

      IF compressorState = 1 THEN
        compressor := TRUE;
      ELSE
        compressor := FALSE;
      END_IF;

      IF gstState = 1 THEN
        gstSig := TRUE;
      ELSE
        gstSig := FALSE;
      END_IF;
      (* ELSE System running in manual mode *)
    END_IF;
  (* System stop state *)
  ELSE
    compressorState := 0;
    compressor := FALSE;
    systemValve := FALSE;
    gstState := 0;
    gstSig := FALSE;
  END_IF;

  (* Increase the counters *)
  countHeartbeat := countHeartbeat + 1;
END_PROGRAM

CONFIGURATION Config0
  RESOURCE Res0 ON PLC
    TASK TaskMain(INTERVAL := T#50ms,PRIORITY := 0);
    PROGRAM Inst0 WITH TaskMain : cybICS;
  END_RESOURCE
END_CONFIGURATION

(* ---- lb_claude_assisted_206a4fbb8703_0021.st ---- *)
PROGRAM program0
  VAR
    VoltageChk AT %IX0.0 : BOOL := 0;
    Sensor AT %IX0.1 : BOOL;
    Turbine AT %QX10 : BOOL := 0;
    Trip AT %QX0.0 : BOOL := 0;
    Fault AT %QX0.1 : BOOL := 0;
    FaultLight AT %QX0.4 : BOOL := 0;
    Reset AT %QX0.6 : BOOL := 0;
    Teleruptor AT %QW15 : INT := 0;
  END_VAR
  VAR
    Ttime : TIME;
    CTU0 : CTU;
    TOF0 : TOF;
    R_TRIG1 : R_TRIG;
    _TMP_EQ49_OUT : BOOL;
  END_VAR

  Trip := Fault;
  Turbine := NOT(Trip) AND VoltageChk;
  VoltageChk := Sensor;
  R_TRIG1(CLK := Fault);
  CTU0(CU := R_TRIG1.Q, R := Reset, PV := 3);
  Trip := CTU0.Q;
  TOF0(IN := Fault, PT := T# 15000ms);
  FaultLight := TOF0.Q;
  Teleruptor := CTU0.CV;
  _TMP_EQ49_OUT := EQ(Ttime, T# 15000ms);
  Reset := _TMP_EQ49_OUT;
  Ttime := TOF0.ET;
END_PROGRAM

CONFIGURATION Config0

  RESOURCE Res0 ON PLC
    TASK task0(INTERVAL := T#20ms,PRIORITY := 0);
    PROGRAM instance0 WITH task0 : program0;
  END_RESOURCE
END_CONFIGURATION

(* ---- lb_claude_assisted_36932d655e9b_0068.st ---- *)
FUNCTION MID3:REAL

	VAR_INPUT
		IN1 :	REAL;
		IN2 :	REAL;
		IN3 :	REAL;
	END_VAR

	VAR
		_IN1 :	REAL;
		_IN2 :	REAL;
		_IN3 :	REAL;
	END_VAR

	_IN1 := IN1;
	_IN2 := IN2;
	_IN3 := IN3;

	IF _IN1 > _IN2 THEN MID3 := _IN1; _IN1 := _IN2; _IN2 := MID3; END_IF;
	IF _IN2 > _IN3 THEN _IN2 := _IN3; END_IF;
	MID3 := SEL(_IN1 > _IN2, _IN2, _IN1);

END_FUNCTION

FUNCTION _BYTE_TO_INT:INT
	VAR_INPUT
		IN :	BYTE;
	END_VAR

	_BYTE_TO_INT := USINT_TO_INT(BYTE_TO_USINT(IN));
END_FUNCTION

FUNCTION MULTI_IN:REAL

	VAR_INPUT
		IN_1 :	REAL;
		IN_2 :	REAL;
		IN_3 :	REAL;
		DEFAULT :	REAL;
		IN_MIN :	REAL;
		IN_MAX :	REAL;
		MODE :	BYTE;
	END_VAR

	VAR
		count :	INT;
		F1 :	BOOL;
		F2 :	BOOL;
		F3 :	BOOL;
	END_VAR

	F1 :=  in_1 > in_min AND in_1 < in_max;
	F2 :=  in_2 > in_min AND in_2 < in_max;
	F3 :=  in_3 > in_min AND in_3 < in_max;

	CASE _BYTE_TO_INT(mode) OF
	0:	count := 0;
		IF F1 THEN
			count := count + 1;
			MULTI_IN := in_1;
		ELSE
			MULTI_IN := 0.0;
		END_IF;
		IF F2 THEN
			count := count + 1;
			MULTI_IN := MULTI_IN + in_2;
		END_IF;
		IF F3 THEN
			count := count + 1;
			MULTI_IN := MULTI_IN + in_3;
		END_IF;
		MULTI_IN := SEL_REAL(count = 0, MULTI_IN / INT_TO_REAL(count), default);

	1:	MULTI_IN := SEL_REAL(F1, default, IN_1);

	2:	MULTI_IN := SEL_REAL(F2, default, IN_2);

	3:	MULTI_IN := SEL_REAL(F3, default, IN_3);

	4:	MULTI_IN := default;

	5:	MULTI_IN := SEL_REAL(F1, in_max, IN_1);
		IF F2 AND in_2 < MULTI_IN THEN MULTI_IN := in_2; END_IF;
		IF F3 AND in_3 < MULTI_IN THEN MULTI_IN := in_3; END_IF;
		IF MULTI_IN = in_max THEN MULTI_IN := default; END_IF;

	6:	MULTI_IN := SEL_REAL(F1, in_min, IN_1);
		IF F2 AND in_2 > MULTI_IN THEN MULTI_IN := in_2; END_IF;
		IF F3 AND in_3 > MULTI_IN THEN MULTI_IN := in_3; END_IF;
		IF MULTI_IN = in_min THEN MULTI_IN := default; END_IF;

	7:	IF F1 AND F2 AND F3 THEN MULTI_IN := MID3(in_1, in_2, in_3);
		ELSIF F1 AND F2 THEN MULTI_IN := MIN(in_1, in_2);
		ELSIF F1 AND F3 THEN MULTI_IN := MIN(in_1, in_3);
		ELSIF F2 AND F3 THEN MULTI_IN := MIN(in_2, in_3);
		ELSIF F1 THEN MULTI_IN := in_1;
		ELSIF F2 THEN MULTI_IN := in_2;
		ELSIF F3 THEN MULTI_IN := in_3;
		ELSE MULTI_IN := default;
		END_IF;

	END_CASE;

END_FUNCTION

PROGRAM program0
	VAR
		IN_1 :	REAL;
		IN_2 :	REAL;
		IN_3 :	REAL;
		DEFAULT :	REAL;
		IN_MIN :	REAL;
		IN_MAX :	REAL;
		MODE :	BYTE;

		OUT : REAL;
	END_VAR

	OUT := MULTI_IN(IN_1, IN_2, IN_3, DEFAULT, IN_MIN, IN_MAX, MODE);

END_PROGRAM

CONFIGURATION Config0

	RESOURCE Res0 ON PLC
		TASK task0(INTERVAL := T#20ms,PRIORITY := 0);
		PROGRAM instance0 WITH task0 : program0;
	END_RESOURCE

END_CONFIGURATION

(* ---- lb_claude_assisted_3a860dafcf23_0009.st ---- *)
FUNCTION TEMP_NI : REAL
  VAR_INPUT
    RES : REAL;
    R0 : REAL;
  END_VAR

  TEMP_NI := (SQRT(0.30085225 - 2.66E-3 * (R0 - Res)) - 0.5485) * 751.8796992;

  (* From OSCAT Library, www.oscat.de *)
END_FUNCTION

FUNCTION RES_PT : REAL
  VAR_INPUT
    _T : REAL;
    R0 : REAL;
  END_VAR
  VAR
    T2 : REAL;
  END_VAR

  T2 := _T * _T;

  IF _T >= 0.0 THEN
  	RES_PT := R0 * ( 1.0 + 3.90802E-3 * _T + -5.802E-7 * T2);
  ELSE
  	RES_PT := R0 * ( 1.0 + 3.90802E-3 * _T + -5.802E-7 * T2 + -4.27350E-12 * (_T - 100.0) * T2 * _T);
  END_IF;

  (* From OSCAT Library, www.oscat.de *)
END_FUNCTION

FUNCTION TEMP_PT : REAL
  VAR_INPUT
    RES : REAL;
    R0 : REAL;
  END_VAR
  VAR
    _step : REAL := 50.0;
    X : REAL;
    Y : REAL;
    t1 : REAL;
  END_VAR

  X := 3.9083E-3 * R0;
  Y := -5.775E-7 * R0;
  IF Res >= R0 THEN
  	t1 := X * X - 4.0 * Y * (R0 - Res);
  	IF t1 < 0.0 THEN
  		TEMP_PT := 10000.0;
  	ELSE
  		TEMP_PT := (-X + SQRT(t1)) / (2.0 * Y);
  	END_IF;
  ELSE
  	(* since the formula cannot be solved this is a successive approximation *)
  	TEMP_PT := -100.0;
  	WHILE _step > 0.01 DO
  		(* test if result greater or less *)
  		IF RES_PT(TEMP_PT, R0) < res THEN TEMP_PT := TEMP_PT + _step; ELSE TEMP_PT := TEMP_PT - _step; END_IF;
  		_step := _step * 0.5;
  	END_WHILE;
  END_IF;

  (* From OSCAT Library, www.oscat.de *)
END_FUNCTION

FUNCTION MID3 : REAL
  VAR_INPUT
    IN1 : REAL;
    IN2 : REAL;
    IN3 : REAL;
  END_VAR
  VAR
    _IN1 : REAL;
    _IN2 : REAL;
    _IN3 : REAL;
  END_VAR

  _IN1 := IN1; (* VAR_INPUT auf Variablen umkopieren , da diese schreibgeschützt sind *)
  _IN2 := IN2;
  _IN3 := IN3;

  IF _IN1 > _IN2 THEN MID3 := _IN1; _IN1 := _IN2; _IN2 := MID3; END_IF;
  IF _IN2 > _IN3 THEN _IN2 := _IN3; END_IF;
  MID3 := SEL(_IN1 > _IN2, _IN2, _IN1);
  (* from OSCAT library; www.oscat.de  *)
END_FUNCTION

FUNCTION MULTI_IN : REAL
  VAR_INPUT
    IN_1 : REAL;
    IN_2 : REAL;
    IN_3 : REAL;
    DEFAULT : REAL;
    IN_MIN : REAL;
    IN_MAX : REAL;
    MODE : BYTE;
  END_VAR
  VAR
    count : INT;
    F1 : BOOL;
    F2 : BOOL;
    F3 : BOOL;
  END_VAR

  F1 :=  in_1 > in_min AND in_1 < in_max;
  F2 :=  in_2 > in_min AND in_2 < in_max;
  F3 :=  in_3 > in_min AND in_3 < in_max;

  CASE BYTE_TO_INT(mode) OF
  0:	count := 0;
  	IF F1 THEN
  		count := count + 1;
  		MULTI_IN := in_1;
  	ELSE
  		MULTI_IN := 0.0;
  	END_IF;
  	IF F2 THEN
  		count := count + 1;
  		MULTI_IN := MULTI_IN + in_2;
  	END_IF;
  	IF F3 THEN
  		count := count + 1;
  		MULTI_IN := MULTI_IN + in_3;
  	END_IF;
  	MULTI_IN := SEL(count = 0, MULTI_IN / INT_TO_REAL(count), default);

  1:	MULTI_IN := SEL(F1, default, IN_1);

  2:	MULTI_IN := SEL(F2, default, IN_2);

  3:	MULTI_IN := SEL(F3, default, IN_3);

  4:	MULTI_IN := default;

  5:	MULTI_IN := SEL(F1, in_max, IN_1);
  	IF F2 AND in_2 < MULTI_IN THEN MULTI_IN := in_2; END_IF;
  	IF F3 AND in_3 < MULTI_IN THEN MULTI_IN := in_3; END_IF;
  	IF MULTI_IN = in_max THEN MULTI_IN := default; END_IF;

  6:	MULTI_IN := SEL(F1, in_min, IN_1);
  	IF F2 AND in_2 > MULTI_IN THEN MULTI_IN := in_2; END_IF;
  	IF F3 AND in_3 > MULTI_IN THEN MULTI_IN := in_3; END_IF;
  	IF MULTI_IN = in_min THEN MULTI_IN := default; END_IF;

  7:	IF F1 AND F2 AND F3 THEN MULTI_IN := MID3(in_1, in_2, in_3);
  	ELSIF F1 AND F2 THEN MULTI_IN := MIN(in_1, in_2);
  	ELSIF F1 AND F3 THEN MULTI_IN := MIN(in_1, in_3);
  	ELSIF F2 AND F3 THEN MULTI_IN := MIN(in_2, in_3);
  	ELSIF F1 THEN MULTI_IN := in_1;
  	ELSIF F2 THEN MULTI_IN := in_2;
  	ELSIF F3 THEN MULTI_IN := in_3;
  	ELSE MULTI_IN := default;
  	END_IF;

  END_CASE;

  (* From OSCAT Library, www.oscat.de *)
  (* MID3 required *)
END_FUNCTION

PROGRAM program0
  VAR
    LocalVar0 : DINT;
    LocalVar1 : DINT;
    LocalVar2 : DINT;
    ADD1_OUT : DINT;
  END_VAR

  ADD1_OUT := ADD(LocalVar0, LocalVar1);
  LocalVar2 := ADD1_OUT;
END_PROGRAM

FUNCTION TEMP_SI : REAL
  VAR_INPUT
    RES : REAL;
    _RS : REAL;
    TS : REAL;
  END_VAR

  TEMP_SI := (-7.64E-3 + SQRT(Res/_RS* 6.64E-5 - 0.803E-5)) * 30120.48193 + TS;

  (* From OSCAT Library, www.oscat.de *)
END_FUNCTION

FUNCTION RES_NI : REAL
  VAR_INPUT
    _T : REAL;
    R0 : REAL;
  END_VAR
  VAR
    T2 : REAL;
  END_VAR

  T2 := _T*_T;
  Res_NI := R0 + 0.5485*_T + 0.665E-3*T2 + 2.805E-9*T2*T2;

  (* From OSCAT Library, www.oscat.de *)
END_FUNCTION

FUNCTION RES_NTC : REAL
  VAR_INPUT
    _T : REAL;
    RN : REAL;
    B : REAL;
  END_VAR

  RES_NTC := RN * EXP(B * (1.0 / (_T+273.15) - 0.00335401643468053));

  (* From OSCAT Library, www.oscat.de *)
END_FUNCTION

FUNCTION TEMP_NTC : REAL
  VAR_INPUT
    RES : REAL;
    RN : REAL;
    B : REAL;
  END_VAR

  IF res > 0.0 THEN
  	TEMP_NTC := B * 298.15 / (B + LN(RES / RN) * 298.15) -273.15;
  END_IF;

  (* From OSCAT Library, www.oscat.de *)
END_FUNCTION

FUNCTION SENSOR_INT : REAL
  VAR_INPUT
    VOLTAGE : REAL;
    CURRENT : REAL;
    RP : REAL;
    _RS : REAL;
  END_VAR
  VAR
    RG : REAL;
  END_VAR

  IF current <> 0.0 THEN
  	RG := voltage / current;
  	SENSOR_INT := RP * ( RG - _RS) / ( RP + _RS - RG);
  END_IF;

  (* From OSCAT Library, www.oscat.de *)
END_FUNCTION

FUNCTION RES_SI : REAL
  VAR_INPUT
    _T : REAL;
    _RS : REAL;
    TS : REAL;
  END_VAR
  VAR
    TX : REAL;
  END_VAR

  TX := _T - TS;
  RES_SI := _RS * ( 1.0 + 7.64E-3 * TX + 1.66E-5 * TX * TX);

  (* From OSCAT Library, www.oscat.de *)
END_FUNCTION

CONFIGURATION Config0

  RESOURCE Res0 ON PLC
    TASK task0(INTERVAL := T#20ms,PRIORITY := 0);
    PROGRAM instance0 WITH task0 : program0;
  END_RESOURCE
END_CONFIGURATION

(* ---- lb_claude_assisted_48d36cd5c79b_0013.st ---- *)
PROGRAM AutomatedTrafficControl
VAR
    currentTime AT %IW0.0 : INT;        (* Current time in hours (24-hour format) *)
    trafficCondition AT %IW0.1 : INT;   (* Traffic condition (1 for low, 2 for moderate, 3 for high) *)
    trafficLightState AT %QW0.0 : INT;     (* State of the traffic lights (0 for Red", 1 for Green, 2 for Yellow) *)
END_VAR

(* Logical Bug: Incorrect handling of traffic light states in case statement *)
CASE currentTime OF
    0..5: (* Late night *)
        trafficLightState := 2; (* Yellow *)
    6..9: (* Morning rush hour *)
        IF trafficCondition = 3 THEN
            trafficLightState := 1; (* Green *)
        ELSE
            trafficLightState := 0; (* Red *)
        END_IF;
    10..15: (* Day time *)
        trafficLightState := 1; (* Green *)
    16..19: (* Evening rush hour *)
        (* Bug: Red light during high traffic in the evening rush hour *)
        IF trafficCondition = 3 THEN
            trafficLightState := 0; (* Red *)
        ELSE
            trafficLightState := 1; (* Green *)
        END_IF;
    20..23: (* Night *)
        trafficLightState := 2; (* Yellow *)
END_CASE;

(* SetTrafficLightState(trafficLightState); *)
END_PROGRAM

CONFIGURATION STD_CONF

  RESOURCE STD_RESSOURCE ON PLC
    TASK TaskMain(INTERVAL := T#50ms,PRIORITY := 0);
    PROGRAM Inst0 WITH TaskMain : AutomatedTrafficControl;
  END_RESOURCE
END_CONFIGURATION

(* ---- lb_claude_assisted_56b8d5883561_0043.st ---- *)
PROGRAM Cell3
  VAR
    C2_IR AT %IX0.3 : BOOL := true;
    M2_IR AT %IX0.4 : BOOL := true;
    Main AT %IX0.6 : BOOL := true;
    M2_motor AT %QX0.2 : BOOL := true;
    C3_motor AT %QX0.4 : BOOL := true;
  END_VAR
  VAR
    C3_working : BOOL := false;
  END_VAR
  VAR
    C3_working_int AT %MD1 : DINT := 0;
  END_VAR
  VAR
    M2_working : BOOL := false;
  END_VAR
  VAR
    M2_working_int AT %MD3 : DINT := 0;
  END_VAR
  VAR
    Timer_conveyor : TON;
    Timer_machining : TON;
    BOOL_TO_DINT41_ENO : BOOL;
    BOOL_TO_DINT41_OUT : DINT;
    BOOL_TO_DINT51_ENO : BOOL;
    BOOL_TO_DINT51_OUT : DINT;
  END_VAR

  IF NOT(C2_IR) THEN
    C3_working := TRUE; (*set*)
  END_IF;
  C3_motor := NOT(C3_working AND NOT(Main));
  IF NOT(M2_IR) AND C3_working THEN
    M2_working := TRUE; (*set*)
  END_IF;
  IF NOT(M2_IR) AND C3_working THEN
    C3_working := FALSE; (*reset*)
  END_IF;
  M2_motor := NOT(M2_working AND NOT(Main));
  Timer_machining(IN := M2_working, PT := T#3000ms);
  IF Timer_machining.Q THEN
    C3_working := TRUE; (*set*)
  END_IF;
  IF Timer_machining.Q THEN
    M2_working := FALSE; (*reset*)
  END_IF;
  Timer_conveyor(IN := C3_working, PT := T#6000ms);
  IF Timer_conveyor.Q THEN
    C3_working := FALSE; (*reset*)
  END_IF;
  BOOL_TO_DINT41_OUT := BOOL_TO_DINT(EN := TRUE, IN := C3_working, ENO => BOOL_TO_DINT41_ENO);
  C3_working_int := BOOL_TO_DINT41_OUT;
  BOOL_TO_DINT51_OUT := BOOL_TO_DINT(EN := TRUE, IN := M2_working, ENO => BOOL_TO_DINT51_ENO);
  M2_working_int := BOOL_TO_DINT51_OUT;
END_PROGRAM

CONFIGURATION Config0

  RESOURCE Res0 ON PLC
    TASK TaskMain(INTERVAL := T#50ms,PRIORITY := 0);
    PROGRAM Inst0 WITH TaskMain : Cell3;
  END_RESOURCE
END_CONFIGURATION

(* ---- lb_claude_assisted_58d6ea93ad17_0022.st ---- *)
PROGRAM Cell2
  VAR
    C1_IR AT %IX0.3 : BOOL := true;
    M1_IR AT %IX0.4 : BOOL := true;
    Main AT %IX0.6 : BOOL := true;
    M1_motor AT %QX0.2 : BOOL := true;
    C2_motor AT %QX0.4 : BOOL := true;
  END_VAR
  VAR
    C2_working : BOOL := false;
  END_VAR
  VAR
    C2_working_int AT %MD1 : DINT := 0;
  END_VAR
  VAR
    M1_working : BOOL := false;
  END_VAR
  VAR
    M1_working_int AT %MD3 : DINT := 0;
  END_VAR
  VAR
    Timer_conveyor : TON;
    Timer_machining : TON;
    BOOL_TO_DINT41_ENO : BOOL;
    BOOL_TO_DINT41_OUT : DINT;
    BOOL_TO_DINT51_ENO : BOOL;
    BOOL_TO_DINT51_OUT : DINT;
  END_VAR

  IF NOT(C1_IR) THEN
    C2_working := TRUE; (*set*)
  END_IF;
  C2_motor := NOT(C2_working AND NOT(Main));
  IF NOT(M1_IR) AND C2_working THEN
    M1_working := TRUE; (*set*)
  END_IF;
  IF NOT(M1_IR) AND C2_working THEN
    C2_working := FALSE; (*reset*)
  END_IF;
  M1_motor := NOT(M1_working AND NOT(Main));
  Timer_machining(IN := M1_working, PT := T#3000ms);
  IF Timer_machining.Q THEN
    C2_working := TRUE; (*set*)
  END_IF;
  IF Timer_machining.Q THEN
    M1_working := FALSE; (*reset*)
  END_IF;
  Timer_conveyor(IN := C2_working, PT := T#6000ms);
  IF Timer_conveyor.Q THEN
    C2_working := FALSE; (*reset*)
  END_IF;
  BOOL_TO_DINT41_OUT := BOOL_TO_DINT(EN := TRUE, IN := C2_working, ENO => BOOL_TO_DINT41_ENO);
  C2_working_int := BOOL_TO_DINT41_OUT;
  BOOL_TO_DINT51_OUT := BOOL_TO_DINT(EN := TRUE, IN := M1_working, ENO => BOOL_TO_DINT51_ENO);
  M1_working_int := BOOL_TO_DINT51_OUT;
END_PROGRAM

CONFIGURATION Config0

  RESOURCE Res0 ON PLC
    TASK TaskMain(INTERVAL := T#50ms,PRIORITY := 0);
    PROGRAM Inst0 WITH TaskMain : Cell2;
  END_RESOURCE
END_CONFIGURATION
